END_VAR
M_Read := THIS^.stSeqCtrlGeneral.eActiveSeqState = E_SEQ_GENERAL.DONE;

// Assign input
THIS^.udiDBID := udiDBID;
THIS^.sTableName := sTableName;
THIS^.sDBSymbolName := sDBSymbolName;
THIS^.eOrderBy := eOrderBy;
THIS^.eOrderType := eOrderType;
THIS^.nStartIndex := nStartIndex;
THIS^.nRecordCount := nRecordCount;
THIS^.pData2 := pData2;
THIS^.cbData := cbData;

// General
IF THIS^.stSeqCtrlGeneral.eActiveSeqState = E_SEQ_GENERAL.READY THEN
  THIS^.eNextSeq := E_SEQ_DATABASE.READ;
  THIS^.stSeqCtrlGeneral.eActiveSeqState := E_SEQ_GENERAL.EXECUTE;
END_IF

// Example
(*
VAR
    fbPLCDBRead    : FB_PLCDBReadEvt (sNetID := '', tTimeout := T#5S);
    ReadStruct     : ST_StandardRecord;
    tcMessage      : I_TcMessage;
END_VAR

------------------------------------------------------------------------

IF fbPLCDBRead.Read(
    hDBID:= 1, 
    sTableName:= 'MyTable_WithLReal', 
    sDBSymbolName:= 'MyValue', 
    eOrderBy:= E_OrderColumn.ID, 
    eOrderType:= E_OrderType.DESC, 
    nStartIndex:= 0, 
    nRecordCount:= 1, 
    pData:= ADR(ReadStruct), 
    cbData:= SIZEOF(ReadStruct))
THEN
    IF fbPLCDBRead.bError THEN
        tcMessage := fbPLCDBRead.ipTcResult;
        nState := 255; 
    ELSE
        nState := 0;
    END_IF
END_IF
*)
END_METHOD

METHOD M_ReadStruct : BOOL

VAR_INPUT
  /// Indicates the ID of the database to be used.
  udiDBID:                    UDINT;
  /// Name of the table that is to be read.
  sTableName:                 T_MaxString;
  /// Address of the array containing the column name to be read.
  pColumnNames:               POINTER TO ARRAY [0..MAX_DBCOLUMNS] OF STRING(50);
  /// Length of the column name array
  cbColumnNames:              UDINT;
  /// Name the sorting column
  sOrderByColumn:             STRING(50);
  /// Sorting direction (ASC or DESC)
  eOrderType:                 E_OrderType;
  /// Indicates the index of the first record to be read.
  nStartIndex:                UDINT;
  /// Indicates the number of records to be read.
  nRecordCount:               UDINT;
  /// Address of the structure array into which the records are to be written.
  pData:                      POINTER TO BYTE;
  /// Indicates the size of the structure array in bytes.
  cbData:                     UDINT;
END_VAR
VAR
  
END_VAR
M_ReadStruct := THIS^.stSeqCtrlGeneral.eActiveSeqState = E_SEQ_GENERAL.DONE;

// Assign input
THIS^.udiDBID := udiDBID;
THIS^.sTableName := sTableName;
THIS^.pColumnNames := pColumnNames;
THIS^.cbColumnNames := cbColumnNames;
THIS^.sOrderByColumn := sOrderByColumn;
THIS^.eOrderType := eOrderType;
THIS^.nStartIndex := nStartIndex;
THIS^.nRecordCount := nRecordCount;
THIS^.pData := pData;
THIS^.cbData := cbData;

// General
IF THIS^.stSeqCtrlGeneral.eActiveSeqState = E_SEQ_GENERAL.READY THEN
  THIS^.eNextSeq := E_SEQ_DATABASE.READ_STRUCT;
  THIS^.stSeqCtrlGeneral.eActiveSeqState := E_SEQ_GENERAL.EXECUTE;
END_IF

// Example
(*
VAR
    fbPLCDBRead    : FB_PLCDBReadEvt (sNetID := '', tTimeout := T#5S);
    myCustomStruct : ST_Record;
    tcMessage      : I_TcMessage;
END_VAR

------------------------------------------------------------------------

TYPE ST_Record :
STRUCT
    nID        : LINT;
    dtTimestamp: DATE_AND_TIME;
    sName      : STRING;
    nSensor1   : LREAL;
    nSensor2   : LREAL;
END_STRUCT
END_TYPE

--------------------------------------------------------------------------

// set columnnames
ColumnNames[0] := 'ID';
ColumnNames[1] := 'Timestamp';
ColumnNames[2] := 'Name';
ColumnNames[3] := 'Sensor1';
ColumnNames[4] := 'Sensor2';

IF fbPLCDBRead.ReadStruct(
    hDBID:= 1, 
    sTableName:= 'MyTable_Struct', 
    pColumnNames:= ADR(ColumnNames), 
    cbColumnNames:= SIZEOF(ColumnNames), 
    sOrderByColumn:= ColumnNames[0], 
    eOrderType:= E_OrderType.DESC, 
    nStartIndex:= 0, 
    nRecordCount:= 1, 
    pData:= ADR(myCustomStruct), 
    cbData:= SIZEOF(myCustomStruct))
THEN
    IF fbPLCDBRead.bError THEN
        tcMessage:= fbPLCDBRead.ipTcResult;
        nState := 255; 
    ELSE
        nState := 0;
    END_IF
END_IF
*)
END_METHOD

METHOD M_Reset : BOOL
M_Reset := THIS^.stSeqCtrlGeneral.eActiveSeqState = E_SEQ_GENERAL.DONE;

// General
IF THIS^.stSeqCtrlGeneral.eActiveSeqState = E_SEQ_GENERAL.READY THEN
  THIS^.eNextSeq := E_SEQ_DATABASE.INIT;
  THIS^.stSeqCtrlGeneral.eActiveSeqState := E_SEQ_GENERAL.EXECUTE;
END_IF
END_METHOD

(*=== Method: M_Run  ============================================

 @brief: Here is the global code (Timer, Event, Flange,...)*)
METHOD M_Run
END_METHOD

METHOD M_SetReady : BOOL
VAR_INPUT
END_VAR
M_SetReady := TRUE
              AND THIS^.stSeqCtrlGeneral.eActiveSeqState = E_SEQ_GENERAL.READY
              AND THIS^.eSeq = E_SEQ_DATABASE.BASE;

THIS^.stSeqCtrlGeneral.eActiveSeqState := E_SEQ_GENERAL.READY;
THIS^.eNextSeq := E_SEQ_DATABASE.BASE;
END_METHOD

METHOD M_TableExistCheck : BOOL
VAR_INPUT
  /// Indicates the ID of the database to be used.
  udiDBID:                    UDINT;
  /// Name of the table that is to be read.
  sTableName:                 T_MaxString;
END_VAR
VAR_OUTPUT
  /// Result
  bResult:                    BOOL;
END_VAR
M_TableExistCheck := THIS^.stSeqCtrlGeneral.eActiveSeqState = E_SEQ_GENERAL.DONE;

// Assign input
THIS^.udiDBID := udiDBID;
THIS^.sTableName := sTableName;
THIS^.sCmd := CONCAT('SELECT * FROM $'', sTableName);
THIS^.sCmd := CONCAT(THIS^.sCmd, '$'');
THIS^.pSQLCmd := ADR(THIS^.sCmd);
THIS^.cbSQLCmd := SIZEOF(THIS^.sCmd);

// Assign output
bResult := THIS^.bResult;

// General
IF THIS^.stSeqCtrlGeneral.eActiveSeqState = E_SEQ_GENERAL.READY THEN
  THIS^.eNextSeq := E_SEQ_DATABASE.TABLE_EXIST_CHECK;
  THIS^.stSeqCtrlGeneral.eActiveSeqState := E_SEQ_GENERAL.EXECUTE;
END_IF
END_METHOD

METHOD M_Write : BOOL

VAR_INPUT
  /// Indicates the ID of the database to be used.
  udiDBID:            UDINT;
  /// Name of the table that is to be write.
  sTableName:         T_MaxString;
  /// Address of the variable to be logged in the standard table structure.
  pValue:             POINTER TO BYTE;
  /// Length of the variable to be logged.
  cbValue:            UDINT;
  /// Name that is logged in the table.
  sDBSymbolName:      STRING;
  /// Indicates the write mode. (append, update, ring buffer)
  eDBWriteMode:       E_WriteMode;
  /// Additional parameter(s) for the "ring buffer" write mode.
  nRingBuffParameter: UDINT;
END_VAR
M_Write := THIS^.stSeqCtrlGeneral.eActiveSeqState = E_SEQ_GENERAL.DONE;

// Assign input
THIS^.udiDBID := udiDBID;
THIS^.sTableName := sTableName;
THIS^.pValue := pValue;
THIS^.cbValue := cbValue;
THIS^.sDBSymbolName := sDBSymbolName;
THIS^.eDBWriteMode := eDBWriteMode;
THIS^.nRingBuffParameter := nRingBuffParameter;

// General
IF THIS^.stSeqCtrlGeneral.eActiveSeqState = E_SEQ_GENERAL.READY THEN
  THIS^.eNextSeq := E_SEQ_DATABASE.WRITE;
  THIS^.stSeqCtrlGeneral.eActiveSeqState := E_SEQ_GENERAL.EXECUTE;
END_IF

// Example
(*
VAR
    fbPLCDBWrite    : FB_PLCDBWriteEvt(sNetID := '', tTimeout := T#5S);
    myValue         : LREAL := 43.23;
    tcMessage       : I_TcMessage;
END_VAR

------------------------------------------------------------------------

IF fbPLCDBWrite.Write(
    hDBID:= 1, 
    sTableName:= 'myTable_WithLReal',
    pValue:= ADR(myValue), 
    cbValue:= SIZEOF(myValue), 
    sDBSymbolName:= 'MyValue', 
    eDBWriteMode:= E_WriteMode.eADS_TO_DB_RingBuff_Count, 
    nRingBuffParameter:= 3) 
THEN
    IF fbPLCDBWrite.bError THEN
        tcMessage := fbPLCDBWrite.ipTcResult;
        nState := 255; 
    ELSE
        nState := 0; 
    END_IF
END_IF
*)
END_METHOD

METHOD M_WriteBySymbol : BOOL

VAR_INPUT
  /// Indicates the ID of the database to be used.
  udiDBID:            UDINT;
  /// Name of the table that is to be write.
  sTableName:         T_MaxString;
  /// ADS device from which a symbol is to be logged in the standard table structure.
  stADSDevice:        ST_ADSDevice;
  /// Symbol name of the variable to be written
  stSymbol:           ST_Symbol;
  /// Indicates the write mode. (append, update, ring buffer)
  eDBWriteMode:       E_WriteMode;
  /// Additional parameter(s) for the "ring buffer" write mode.
  nRingBuffParameter: UDINT;
END_VAR
M_WriteBySymbol := THIS^.stSeqCtrlGeneral.eActiveSeqState = E_SEQ_GENERAL.DONE;

// Assign input
THIS^.udiDBID := udiDBID;
THIS^.sTableName := sTableName;
THIS^.stADSDevice := stADSDevice;
THIS^.stSymbol := stSymbol;
THIS^.eDBWriteMode := eDBWriteMode;
THIS^.nRingBuffParameter := nRingBuffParameter;



// General
IF THIS^.stSeqCtrlGeneral.eActiveSeqState = E_SEQ_GENERAL.READY THEN
  THIS^.eNextSeq := E_SEQ_DATABASE.WRITE_BY_SYMBOL;
  THIS^.stSeqCtrlGeneral.eActiveSeqState := E_SEQ_GENERAL.EXECUTE;
END_IF

// Example
(*
VAR
    fbPLCDBWrite    :  FB_PLCDBWriteEvt(sNetID := '', tTimeout := T#5S);
    myValue         :  LREAL := 43.23;
    myAdsDevice     :  ST_ADSDevice;
    mySymbol        :  ST_Symbol;
    tcMessage       :  I_TcMessage;
END_VAR

------------------------------------------------------------------------

// Set ADSDevice Information
myAdsDevice.sDevNetID     := '127.0.0.1.1.1';
myAdsDevice.nDevPort      := 851;
myAdsDevice.eADSRdWrtMode := E_ADSRdWrtMode.bySymbolName; 
myAdsDevice.tTimeout      := T#5S; 

// Set Symbol Information
mySymbol.eDataType        := E_PLCDataType.eType_LREAL;
mySymbol.sDBSymbolName    := 'MySymbol';
mySymbol.sSymbolName      := 'MAIN.myValue';
mySymbol.nBitSize         := 8;

// Call Functionblock
IF fbPLCDBWrite.WriteBySymbol(
    hDBID:= 1, 
    sTableName:= 'myTable_WithLReal', 
    stADSDevice:= myAdsDevice, 
    stSymbol:= mySymbol, 
    eDBWriteMode:= E_WriteMode.eADS_TO_DB_Append, 
    nRingBuffParameter:= 1) 
THEN
    IF fbPLCDBWrite.bError THEN
        tcMessage := fbPLCDBWrite.ipTcResult;
        nState := 255; 
    ELSE
        nState := 0;
    END_IF
END_IF
*)
END_METHOD

METHOD M_WriteStruct : BOOL
VAR_INPUT
  /// Indicates the ID of the database to be used.
  udiDBID:        UDINT;
  /// Name of the table that is to be write.
  sTableName:     T_MaxString;
  /// Address of a structure that is to be logged in a freely selectable table structure.
  pRecord:        POINTER TO BYTE;
  /// Length of the structure to be written
  cbRecord:       UDINT;
  /// Address of the array containing the column name to be filled.
  pColumnNames:   POINTER TO ARRAY [0..MAX_DBCOLUMNS] OF STRING(50);
  /// Length of the column name array
  cbColumnNames:  UDINT;
END_VAR
M_WriteStruct := THIS^.stSeqCtrlGeneral.eActiveSeqState = E_SEQ_GENERAL.DONE;

// Assign input
THIS^.udiDBID := udiDBID;
THIS^.sTableName := sTableName;
THIS^.pRecord := pRecord;
THIS^.cbRecord := cbRecord;
THIS^.pColumnNames := pColumnNames;
THIS^.cbColumnNames := cbColumnNames;

// General
IF THIS^.stSeqCtrlGeneral.eActiveSeqState = E_SEQ_GENERAL.READY THEN
  THIS^.eNextSeq := E_SEQ_DATABASE.WRITE_STRUCT;
  THIS^.stSeqCtrlGeneral.eActiveSeqState := E_SEQ_GENERAL.EXECUTE;
END_IF

// Example
(*
VAR
    fbPLCDBWrite    :  FB_PLCDBWriteEvt(sNetID := '', tTimeout := T#5S);
    myRecord        :  ST_Record;
    ColumnNames     :  ARRAY[0..4] OF STRING(50);
    
    systime         :  GETSYSTEMTIME;
    currentTime     :  T_FILETIME;
    tcMessage       :  I_TcMessage;
END_VAR

------------------------------------------------------------------------

TYPE ST_Record :
STRUCT
    nID        : LINT;
    dtTimestamp: DATE_AND_TIME;
    sName      : STRING;
    nSensor1   : LREAL;
    nSensor2   : LREAL;
END_STRUCT
END_TYPE

------------------------------------------------------------------------

// set Values
systime(timeLoDw => currentTime.dwLowDateTime, timeHiDW => currentTime.dwHighDateTime );
myRecord.dtTimestamp := FILETIME_TO_DT(currentTime);
myRecord.sName       := 'MyStructVal';
myRecord.nSensor1    := 12.34;
myRecord.nSensor2    := 102.5;

// set columnnames
ColumnNames[0] := 'ID';
ColumnNames[1] := 'Timestamp';
ColumnNames[2] := 'Name';
ColumnNames[3] := 'Sensor1';
ColumnNames[4] := 'Sensor2';

// Call Functionblock
IF fbPLCDBWrite.WriteStruct(
    hDBID:= 1, 
    sTableName:= 'myTable_Struct', 
    pRecord:= ADR(myRecord), 
    cbRecord:= SIZEOF(myRecord), 
    pColumnNames:= ADR(ColumnNames) , 
    cbColumnNames:= SIZEOF(ColumnNames))
THEN
    IF fbPLCDBWrite.bError THEN
        tcMessage := fbPLCDBWrite.ipTcResult;
        nState := 255; 
    ELSE
        nState := 0;
    END_IF
END_IF
*)
END_METHOD

PROPERTY P_Connected : BOOL
GET
P_Connected := THIS^.fbSQLDatabase.bConnected;
END_GET
END_PROPERTY

{warning 'Eigenschaftenimplementierung hinzufügen'}
PROPERTY P_Error : BOOL
GET
P_Error := THIS^.stSeqCtrlGeneral.eActiveSeqState = E_SEQ_GENERAL.ERROR;
END_GET
END_PROPERTY

{warning 'Eigenschaftenimplementierung hinzufügen'}
(*=== Property: P_Event  ============================================

 @param [set]: 	Set the Structure "ST_EVENT" from another Object
 @param [get]: 	Return the Structure "ST_EVENT", it contains the actual 
					event of the Object *)
PROPERTY P_Event : GenLib.ST_EVENT
GET
END_GET
SET
END_SET
END_PROPERTY

{warning 'Eigenschaftenimplementierung hinzufügen'}
(*=== Property: P_FullObjectPath  ============================================

 @param [set]: 	Set the Object Path (Clear String of Object)
 @param [get]: 	Return the Objectpath *)
PROPERTY P_FullObjectPath : STRING
GET
P_FullObjectPath:= THIS^.strFullObjectPath;
END_GET
SET
THIS^.strFullObjectPath:=P_FullObjectPath;
END_SET
END_PROPERTY

{warning 'Eigenschaftenimplementierung hinzufügen'}
(*=== Property: P_Global_Ack  ============================================

 @param [set]: 	Set the Bit for Ack from another Object
 @param [get]: 	Return the state of Ack Bit*)
PROPERTY P_Global_Ack : BOOL
GET
END_GET
SET
END_SET
END_PROPERTY

{warning 'Eigenschaftenimplementierung hinzufügen'}
(*=== Property: P_GlobalID  ============================================

 @param [set]: 	-
 @param [get]: 	Return the string of instance path*)
PROPERTY P_GlobalID : STRING
GET
P_GlobalID:= THIS^.strInstancePath;
END_GET
END_PROPERTY

END_FUNCTION_BLOCK

// ---- MODULE/FREQUENCE/POU/FB_FREQENCE.TcPOU
{attribute 'reflection'} 
{attribute 'no_explicit_call' := 'do not call this POU directly'} 
FUNCTION_BLOCK PUBLIC FB_FREQENCE IMPLEMENTS  I_FREQ_GEN
VAR_INPUT
END_VAR
VAR_OUTPUT
END_VAR
VAR
	{attribute 'instance-path'} 
    {attribute 'noinit'} 
	strInstancePath: STRING;
	strFullObjectPath: STRING;
	stEvent: ST_EVENT;
	bAck: BOOL;
	
	iStep:		INT:=0;
	tonLow:		TON;
	tonHigh:	TON;
	tFreq:		TIME;
	bState:		BOOL;
	iFreqence:	INT;
	fTrig:		F_TRIG;
	rTrig:		R_TRIG;
END_VAR

(*=== Method: M_Run  ============================================

 @brief: Here is the global code (Timer, Event, Flange,...)*)
METHOD M_Run
tFreq := TO_TIME(TO_REAL(1000 * iFreqence) / 2);

CASE iStep OF
0:;	IF tonLow.Q THEN iStep := 1; END_IF;
1:;	IF tonHigh.Q THEN iStep := 0; END_IF;
ELSE
	iStep := 0;
END_CASE

tonHigh(IN:=(iStep=1), PT:= tFreq);
tonLow(IN:= (iStep=0), PT:= tFreq);

bState:=(iStep>=1);

fTrig(CLK:=bState);
rTrig(CLK:=bState);
END_METHOD

METHOD M_SetFrequence : bool
VAR_INPUT
	iFreqence: INT;
END_VAR
M_SetFrequence := TRUE;

THIS^.iFreqence := iFreqence;
END_METHOD

(*=== Property: P_Event  ============================================

 @param [set]: 	Set the Structure "ST_EVENT" from another Object
 @param [get]: 	Return the Structure "ST_EVENT", it contains the actual 
					event of the Object *)
PROPERTY P_Event : GenLib.ST_EVENT
GET
P_Event:=stEvent;
END_GET
SET
stEvent:=P_Event;
END_SET
END_PROPERTY

PROPERTY P_FTrig : BOOL
GET
P_FTrig:=THIS^.fTrig.Q;
END_GET
END_PROPERTY

(*=== Property: P_FullObjectPath  ============================================

 @param [set]: 	Set the Object Path (Clear String of Object)
 @param [get]: 	Return the Objectpath *)
PROPERTY P_FullObjectPath : STRING
GET
P_FullObjectPath:= THIS^.strFullObjectPath;
END_GET
SET
THIS^.strFullObjectPath:=P_FullObjectPath;
END_SET
END_PROPERTY

(*=== Property: P_Global_Ack  ============================================

 @param [set]: 	Set the Bit for Ack from another Object
 @param [get]: 	Return the state of Ack Bit*)
PROPERTY P_Global_Ack : BOOL
GET
P_Global_Ack:=THIS^.bAck;
END_GET
SET
THIS^.bAck:=P_Global_Ack;
END_SET
END_PROPERTY

(*=== Property: P_GlobalID  ============================================

 @param [set]: 	-
 @param [get]: 	Return the string of instance path*)
PROPERTY P_GlobalID : STRING
GET
P_GlobalID:= THIS^.strInstancePath;
END_GET
END_PROPERTY

PROPERTY P_RTrig : BOOL
GET
P_RTrig := THIS^.rTrig.Q;
END_GET
END_PROPERTY

PROPERTY P_State : BOOL
GET
P_State:=THIS^.bState;
END_GET
END_PROPERTY

END_FUNCTION_BLOCK

// ---- MODULE/GENERAL/F_Lineare_Regression.TcPOU
FUNCTION F_Lineare_Regression : stRampAnalytic
VAR_IN_OUT
	Messwerte:          ARRAY[*] OF stMesswerte;
	uiStart: 	          UINT;	
	uiEnd: 		          UINT; 	///Bei 0 gilt Upper Bound
END_VAR
VAR
	i: 					        DINT;
	diLow: 				      DINT;
	diHigh: 			      DINT;
	rMittelwert: 		    stMesswerte;
	lrSteigung: 		    LREAL;
	lrAchsenabschnitt: 	LREAL;
	lrTempY_s: 			    LREAL;
	lrZaehlerMw: 		    LREAL;
	lrNennerMw: 		    LREAL;
	lrSumSqrtY_Ys:		  LREAL;
	lrSumSqrtY_Yd:		  LREAL;
	lrSqrtR:			      LREAL;
	
	stOut:				      stRampAnalytic;
	bFault:             BOOL;
END_VAR

F_Lineare_Regression.lrGain := 0;
F_Lineare_Regression.lrOffset := 0;
F_Lineare_Regression.lrExp2R := -1;
diLow := LOWER_BOUND(Messwerte, 1);
diHigh := UPPER_BOUND(Messwerte, 1);
IF uiEnd > 0 THEN
	diLow := uiStart;
	diHigh := uiEnd;
END_IF 
rMittelwert.X := 0;
rMittelwert.Y := 0;
//Mittelwert ermitteln
FOR i := diLow TO diHigh DO
	rMittelwert.X := rMittelwert.X + Messwerte[i].X;
	rMittelwert.Y := rMittelwert.Y + Messwerte[i].Y;
END_FOR
	IF (DINT_TO_REAL(diHigh - diLow) + 1) <> 0 THEN
	rMittelwert.X := rMittelwert.X / (DINT_TO_REAL(diHigh - diLow) + 1);
	rMittelwert.Y := rMittelwert.Y / (DINT_TO_REAL(diHigh - diLow) + 1);
ELSE
	bFault := TRUE;	
END_IF

//Steigung = Mittelwert X durch Mittelwert Y


lrZaehlerMw := 0;
lrNennerMw := 0;

FOR i:=diLow TO diHigh DO
	lrZaehlerMw :=	lrZaehlerMw + (Messwerte[i].X - rMittelwert.X) * (Messwerte[i].Y - rMittelwert.Y);
	//lrNennerMw:=	lrNennerMw+		(basic.expn((Messwerte[i].X-rMittelwert.X),2));
END_FOR
//lrZaehlerMw:=	lrZaehlerMw	/(DINT_TO_REAL(diHigh-diLow)+0);
//lrNennerMw:=	lrNennerMw	/(DINT_TO_REAL(diHigh-diLow)+0);


//Steigung = 
IF lrNennerMw <> 0 THEN
	lrSteigung := lrZaehlerMw / lrNennerMw;
ELSE
	bFault := TRUE;
END_IF
lrAchsenabschnitt := rMittelwert.Y - (lrSteigung * rMittelwert.X);
(*
FOR i:=diLow TO diHigh DO
	lrTempY_s:=					(Messwerte[i].X*lrSteigung)+lrAchsenabschnitt;
	Messwerte[i].sqr_Y_Ys:=		basic.EXPN((Messwerte[i].Y-lrTempY_s),2);
	
	Messwerte[i].SQR_Y_Yd:=		basic.EXPN((Messwerte[i].Y-rMittelwert.Y),2);
END_FOR
*)
lrSumSqrtY_Ys := 0;
lrSumSqrtY_Yd := 0;
(*
FOR i:=diLow TO diHigh DO
	lrSumSqrtY_Ys:=lrSumSqrtY_Ys+Messwerte[i].sqr_Y_Ys;
	lrSumSqrtY_Yd:=lrSumSqrtY_Yd+Messwerte[i].SQR_Y_Yd;
END_FOR
*)
FOR i := diLow TO diHigh DO
	lrTempY_s := (Messwerte[i].X * lrSteigung) + lrAchsenabschnitt;
	//lrSumSqrtY_Ys:=	lrSumSqrtY_Ys+	basic.EXPN((Messwerte[i].Y-lrTempY_s),2);
	
	//lrSumSqrtY_Yd:=	lrSumSqrtY_Yd+	basic.EXPN((Messwerte[i].Y-rMittelwert.Y),2);
END_FOR

IF lrSumSqrtY_Yd <> 0 THEN
	lrSqrtR := 1 - (lrSumSqrtY_Ys / lrSumSqrtY_Yd);
ELSE
	bFault := TRUE;
END_IF
IF NOT bFault THEN
	F_Lineare_Regression.lrGain := lrSteigung;
	F_Lineare_Regression.lrOffset := lrAchsenabschnitt;
	F_Lineare_Regression.lrExp2R := lrSqrtR;
END_IF

END_FUNCTION

// ---- MODULE/GENERAL/F_RangeSetpoint.TcPOU
FUNCTION F_RangeSetpoint : BOOL
VAR_INPUT
	lrSetpoint: LREAL;
	lrActValue: LREAL;
	lrRangePercent: LREAL;
END_VAR
VAR
	lrTempSetpointUp: LREAL;
	lrTempSetpointDown: LREAL;
END_VAR

F_RangeSetpoint:=FALSE;

lrTempSetpointDown:=lrSetpoint-(lrSetpoint*(lrRangePercent/100.0));
lrTempSetpointUp:=lrSetpoint+(lrSetpoint*(lrRangePercent/100.0));

IF (lrActValue>=lrTempSetpointDown) AND (lrActValue<=lrTempSetpointUp) THEN
	F_RangeSetpoint:=TRUE;
END_IF

END_FUNCTION

// ---- MODULE/GENERAL/INPUTS/POU/FB_BINARY_SWITCH_SENS.TcPOU
FUNCTION_BLOCK FB_BINARY_SWITCH_SENS IMPLEMENTS  I_BINARY_SWITCH_SENS
VAR_INPUT
END_VAR
VAR_OUTPUT
END_VAR
VAR
		
	itfOpMode:										I_OP_MODE;
	{attribute 'instance-path'} 
    {attribute 'noinit'} 
	strInstancePath:								STRING;
	strFullObjectPath:								STRING;
	stEvent:										ST_EVENT;
	bAck:											BOOL;
	
	bSwitch 										AT %I*: BOOL;
	bNC:											BOOL;
	fbEventLogger:									FB_TcEventLogger;
	                                				
	strSymName:										STRING;
	iStepCase:										INT;
	strMessage:										STRING;
	bSensingON:										BOOL;
END_VAR

strFullObjectPath:=F_CreateIdString(THIS^);


stEvent.bEventActive:=FALSE;
IF THIS^.bSensingON AND P_Active THEN
	fbEventLogger.GetAlarm(eventClass:= TC_EVENT_CLASSES.TcSystemEventClass,
							nEventID:=1,
							ipSourceInfo:=TRUE,
							fbAlarm:=TRUE);
END_IF



//Überwachung Eingang
CASE iStepCase OF
	
	0://SENSING Deaktiviert
	
	
	1://SENSING Aktiviert
		
		
	
	
	re
END_CASE

METHOD FB_init : BOOL
VAR_INPUT
	bInitRetains : BOOL; // if TRUE, the retain variables are initialized (warm start / cold start)
	bInCopyCode : BOOL;  // if TRUE, the instance afterwards gets moved into the copy code (online change)
	itfOpMode:			I_OP_MODE;
	bInNC: 				BOOL;///NC:=true; NO:= false
	strMessage:			STRING;
	bSensingON:			BOOL;
END_VAR
THIS^.itfOpMode:=	itfOpMode;
THIS^.bNC:=			bInNC;
THIS^.strMessage:=	strMessage;
THIS^.bSensingON:=	bSensingON;
END_METHOD

(*=== Method: M_Run  ============================================

 @brief: Here is the global code (Timer, Event, Flange,...)*)
METHOD M_Run
END_METHOD

METHOD M_START_SENS : BOOL
VAR_INPUT
	bState	: BOOL;
	tDelay	: TIME;
	eEventType	: GenLib.ENUM_EVENT_TYPE;
END_VAR
IF THIS^.iStepCase=0 THEN
	THIS^.iStepCase:=1;
END_IF
END_METHOD

METHOD M_STOP_SENS : BOOL
END_METHOD

PROPERTY P_Active : BOOL
GET
IF bNC THEN
	P_ACTIVE:= NOT bSwitch;
ELSE
	P_ACTIVE:= bSwitch;
END_IF
END_GET
END_PROPERTY

(*=== Property: P_Event  ============================================

 @param [set]: 	Set the Structure "ST_EVENT" from another Object
 @param [get]: 	Return the Structure "ST_EVENT", it contains the actual 
					event of the Object *)
PROPERTY P_Event : GenLib.ST_EVENT
GET
P_Event:=stEvent;
END_GET
SET
stEvent:=P_Event;
END_SET
END_PROPERTY

(*=== Property: P_FullObjectPath  ============================================

 @param [set]: 	Set the Object Path (Clear String of Object)
 @param [get]: 	Return the Objectpath *)
PROPERTY P_FullObjectPath : STRING
GET
P_FullObjectPath:= THIS^.strFullObjectPath;
END_GET
SET
END_SET
END_PROPERTY

(*=== Property: P_Global_Ack  ============================================

 @param [set]: 	Set the Bit for Ack from another Object
 @param [get]: 	Return the state of Ack Bit*)
PROPERTY P_Global_Ack : BOOL
GET
P_Global_Ack:=THIS^.bAck;
END_GET
SET
THIS^.bAck:=P_Global_Ack;
END_SET
END_PROPERTY

{warning 'Eigenschaftenimplementierung hinzufügen'}
(*=== Property: P_GlobalID  ============================================

 @param [set]: 	-
 @param [get]: 	Return the string of instance path*)
PROPERTY P_GlobalID : STRING
GET
P_GlobalID:= THIS^.strInstancePath;
END_GET
END_PROPERTY

PROPERTY P_No_Nc : BOOL
GET
P_No_Nc:= not THIS^.bNC;
END_GET
END_PROPERTY

PROPERTY P_On : BOOL
GET
P_ON:= bSwitch;
END_GET
END_PROPERTY

PROPERTY P_STATE_SENS : BOOL
GET
END_GET
END_PROPERTY

END_FUNCTION_BLOCK

// ---- MODULE/GENERAL/SIMU_ANALOG_IN/FB_SIMU_ANALOG_IN.TcPOU
{attribute 'reflection'} 
FUNCTION_BLOCK FB_SIMU_ANALOG_IN IMPLEMENTS  I_SIMU_ANALOG_IN
VAR_INPUT
END_VAR
VAR_OUTPUT
END_VAR
VAR
	lrSetPoint: LREAL;
	{attribute 'instance-path'} 
    {attribute 'noinit'} 
	strInstancePath: STRING;
	strFullObjectPath: STRING;
END_VAR

{warning 'Methodenimplementierung hinzufügen'}
(*=== Method: M_Run  ============================================

 @brief: Here is the global code (Timer, Event, Flange,...)*)
METHOD M_Run
THIS^.strFullObjectPath:= F_CreateIdString(THIS^);
END_METHOD

{warning 'Eigenschaftenimplementierung hinzufügen'}
(*=== Property: P_Event  ============================================

 @param [set]: 	Set the Structure "ST_EVENT" from another Object
 @param [get]: 	Return the Structure "ST_EVENT", it contains the actual 
					event of the Object *)
PROPERTY P_Event : GenLib.ST_EVENT
GET
END_GET
SET
END_SET
END_PROPERTY

{warning 'Eigenschaftenimplementierung hinzufügen'}
(*=== Property: P_FullObjectPath  ============================================

 @param [set]: 	Set the Object Path (Clear String of Object)
 @param [get]: 	Return the Objectpath *)
PROPERTY P_FullObjectPath : STRING
GET
P_FullObjectPath:= THIS^.strFullObjectPath;
END_GET
SET
THIS^.strFullObjectPath:=P_FullObjectPath;
END_SET
END_PROPERTY

{warning 'Eigenschaftenimplementierung hinzufügen'}
(*=== Property: P_Global_Ack  ============================================

 @param [set]: 	Set the Bit for Ack from another Object
 @param [get]: 	Return the state of Ack Bit*)
PROPERTY P_Global_Ack : BOOL
GET
END_GET
SET
END_SET
END_PROPERTY

{warning 'Eigenschaftenimplementierung hinzufügen'}
(*=== Property: P_GlobalID  ============================================

 @param [set]: 	-
 @param [get]: 	Return the string of instance path*)
PROPERTY P_GlobalID : STRING
GET
P_GlobalID:= THIS^.strInstancePath;
END_GET
END_PROPERTY

{warning 'Eigenschaftenimplementierung hinzufügen'}
PROPERTY P_SETPOINT : LREAL
SET
lrSetPoint:=P_SETPOINT;
END_SET
END_PROPERTY


PROPERTY P_VALUE : LREAL
GET
P_VALUE:=lrSetPoint;
END_GET
END_PROPERTY

END_FUNCTION_BLOCK

// ---- MODULE/HMI/POU/FB_HMI_CTRL.TcPOU
FUNCTION_BLOCK FB_HMI_CTRL IMPLEMENTS I_HMI_CTRL
VAR_INPUT
END_VAR
VAR_OUTPUT
END_VAR
VAR
  strInstancePath:                STRING;
	strFullObjectPath:              STRING;
  strErrorMsg:                    STRING := '';
  bInHP:                          BOOL;
	stEvent:                        ST_EVENT;
	bAck:                           BOOL;
	itfOpMode:			                I_OP_MODE;
  
  //HMI Start
	fbHmiStart:							  NT_StartProcess;
	bHmiStart:							  BOOL;
	//HMI Kill
	fbTaskKill:							  NT_StartProcess;
	bTaskKill:							  BOOL;
	//Shutdown Windows
	fbShutdown:							  NT_StartProcess;
	bShutdown:							  BOOL;
	//Reboot Windows
	fbReboot:							    NT_StartProcess;
	bReboot:							    BOOL;
	//Windows Keyboard
	fbWinKeyboard:						NT_StartProcess;
	bWinKeyboard:						  BOOL;
END_VAR

fbHmiStart(
	NETID:= '', 
	PATHSTR:= 'C:\Program Files (x86)\Microsoft\Edge\Application\msedge.exe', 
	DIRNAME:= 'C:\Program Files (x86)\Microsoft\Edge\Application', 
	COMNDLINE:= '--kiosk http://Administrator:1@127.0.0.1:1010 --edge-kiosk-type=fullscreen', 
	START:= bHmiStart, 
	TMOUT:= T#25S, 
	BUSY=> , 
	ERR=> , 
	ERRID=> );
IF fbHmiStart.BUSY THEN
	bHmiStart:=FALSE;
END_IF

fbTaskKill(
	NETID:= '', 
	PATHSTR:= 'C:\Scripts\CloseHMI.bat', 
	DIRNAME:= 'C:\Scripts', 
	COMNDLINE:= '', 
	START:= bTaskKill, 
	TMOUT:= T#5S, 
	BUSY=> , 
	ERR=> , 
	ERRID=> );
IF fbTaskKill.BUSY THEN
	bTaskKill:=FALSE;
END_IF

fbWinKeyboard(
	NETID:= '', 
	PATHSTR:= 'C:\Scripts\Keyboard.bat', 
	DIRNAME:= 'C:\Scripts', 
	COMNDLINE:= '', 
	START:= bWinKeyboard, 
	TMOUT:= T#5S, 
	BUSY=> , 
	ERR=> , 
	ERRID=> );
IF fbWinKeyboard.BUSY THEN
	bWinKeyboard:=FALSE;
END_IF

fbShutdown(
	NETID:= '', 
	PATHSTR:= 'C:\Scripts\Shutdown.bat', 
	DIRNAME:= 'C:\Scripts', 
	COMNDLINE:= '', 
	START:= bShutdown, 
	TMOUT:= T#30S, 
	BUSY=> , 
	ERR=> , 
	ERRID=> );
IF fbShutdown.BUSY THEN
	bShutdown:=FALSE;
END_IF

fbReboot(
	NETID:= '', 
	PATHSTR:= 'C:\Scripts\Reboot.bat', 
	DIRNAME:= 'C:\Scripts', 
	COMNDLINE:= '', 
	START:= bReboot, 
	TMOUT:= T#30S, 
	BUSY=> , 
	ERR=> , 
	ERRID=> );
IF fbReboot.BUSY THEN
	bReboot:=FALSE;
END_IF

METHOD FB_init : BOOL
VAR_INPUT
	bInitRetains : BOOL; // if TRUE, the retain variables are initialized (warm start / cold start)
	bInCopyCode : BOOL;  // if TRUE, the instance afterwards gets moved into the copy code (online change)
END_VAR
END_METHOD

METHOD M_CloseHMI : BOOL
bTaskKill := TRUE;
END_METHOD

METHOD M_HideWinKeyboard : BOOL
END_METHOD

METHOD M_PCReboot : BOOL
bReboot := TRUE;
END_METHOD

METHOD M_PCShutdown : BOOL
bShutdown := TRUE;
END_METHOD

{warning 'Methodenimplementierung hinzufügen'}
(*=== Method: M_Run  ============================================

 @brief: Here is the global code (Timer, Event, Flange,...)*)
METHOD M_Run
END_METHOD

{warning 'Methodenimplementierung hinzufügen'}
METHOD M_SetReady : BOOL
END_METHOD

METHOD M_ShowWinKeyboard : BOOL
bWinKeyboard := TRUE;
END_METHOD

METHOD M_StartHMI : BOOL
bHmiStart := TRUE;
END_METHOD

{warning 'Eigenschaftenimplementierung hinzufügen'}
PROPERTY P_ErrorMsg : STRING
GET
END_GET
SET
END_SET
END_PROPERTY

{warning 'Eigenschaftenimplementierung hinzufügen'}
(*=== Property: P_Event  ============================================

 @param [set]: 	Set the Structure "ST_EVENT" from another Object
 @param [get]: 	Return the Structure "ST_EVENT", it contains the actual 
					event of the Object *)
PROPERTY P_Event : GenLib.ST_EVENT
GET
END_GET
SET
END_SET
END_PROPERTY

{warning 'Eigenschaftenimplementierung hinzufügen'}
(*=== Property: P_FullObjectPath  ============================================

 @param [set]: 	Set the Object Path (Clear String of Object)
 @param [get]: 	Return the Objectpath *)
PROPERTY P_FullObjectPath : STRING
GET
END_GET
SET
END_SET
END_PROPERTY

{warning 'Eigenschaftenimplementierung hinzufügen'}
(*=== Property: P_Global_Ack  ============================================

 @param [set]: 	Set the Bit for Ack from another Object
 @param [get]: 	Return the state of Ack Bit*)
PROPERTY P_Global_Ack : BOOL
GET
END_GET
SET
END_SET
END_PROPERTY

{warning 'Eigenschaftenimplementierung hinzufügen'}
(*=== Property: P_GlobalID  ============================================

 @param [set]: 	-
 @param [get]: 	Return the string of instance path*)
PROPERTY P_GlobalID : STRING
GET
END_GET
END_PROPERTY

END_FUNCTION_BLOCK

// ---- MODULE/SAFETY/POU/FB_ESTOP.TcPOU
FUNCTION_BLOCK FB_ESTOP IMPLEMENTS I_ESTOP
VAR_INPUT
END_VAR
VAR_OUTPUT
END_VAR
VAR //General
	{attribute 'instance-path'} 
    {attribute 'noinit'} 
	strInstancePath:										STRING;
	strFullObjectPath: 										STRING;
	stEvent: 												ST_EVENT;
	bAck: 													BOOL;
	quitDelayTimer:											TON;

	//Interfaces
	itfOpMode:												I_OP_MODE;
	itfQuitEStop:											I_BINARY_OUTPUT;
	itfEStopLoadingLeftState:								I_BINARY_SWITCH;
	itfEStopLoadingRightState: 								I_BINARY_SWITCH;	
	itfEStopWeighSideState:									I_BINARY_SWITCH;
 
	//Schrittkettensteuerung
	eSeq, eLastSeq, eNextSeq:								E_STEP_STATE_ESTOP:=	E_STEP_STATE_ESTOP.ESTOP_PRESSED;
	tonDelay, tonTimeOut, tonStepTime:						TON;
	tDelay:													TIME := T#100MS;
	tTimeOut:												TIME := T#100MS;
	tTimeOutExt:											TIME := T#100MS;
	bDelayActive, bTimeOutActiveQuit, bTimeOutActiveNoQuit:	BOOL;//Timer Option
	bActiveStep, bDebugAcitve, bDebugNext:					BOOL;//Debug Option
	i:														INT;
    iError:													INT; //ERROR-CODE                    	                   		
	listLastSteps:											ARRAY[0..49] OF ST_LAST_STEPS;	
	strExtraInfo:											STRING; 
	eStep_Type:												E_STEP_STATE_TYPE; 
	bDebugModeActive:										BOOL;   
	bWaitForBreakpoint:										BOOL;
	bBreakpointActive:										BOOL;
	bDebugResume:											BOOL;   
	listBreakpoint:											ARRAY[0..10] OF  INT;  
END_VAR

eLastSeq:=eSeq;

CASE eSeq OF 
E_STEP_STATE_ESTOP.BASE:;
		eSeq:=E_STEP_STATE_ESTOP.ESTOP_OK;
	
E_STEP_STATE_ESTOP.RESET:;
		eSeq:=E_STEP_STATE_ESTOP.BASE;

E_STEP_STATE_ESTOP.ESTOP_OK:;
	IF FALSE
		OR itfEStopLoadingLeftState.P_Active
		OR itfEStopLoadingRightState.P_Active
		OR itfEStopWeighSideState.P_Active
	THEN
		eSeq:=E_STEP_STATE_ESTOP.ESTOP_PRESSED;
	ELSE
		itfOpMode.P_EMERGANCY_STOP:=FALSE;
		eSeq:=E_STEP_STATE_ESTOP.ESTOP_OK;
	END_IF

E_STEP_STATE_ESTOP.ESTOP_PRESSED:;
	IF FALSE
		OR itfEStopLoadingLeftState.P_Active
		OR itfEStopLoadingRightState.P_Active
		OR itfEStopWeighSideState.P_Active
	THEN
		itfOpMode.P_EMERGANCY_STOP:=TRUE;
		eSeq:=E_STEP_STATE_ESTOP.ESTOP_PRESSED;
	ELSE
		eSeq:=E_STEP_STATE_ESTOP.WAIT_QUIT_ESTOP;
	END_IF
					
E_STEP_STATE_ESTOP.WAIT_QUIT_ESTOP:;
	IF itfQuitEStop.P_State THEN
		itfQuitEStop.M_Reset();
	END_IF
	IF FALSE
		OR itfEStopLoadingLeftState.P_Active
		OR itfEStopLoadingRightState.P_Active
		OR itfEStopWeighSideState.P_Active
	THEN
		eSeq:=E_STEP_STATE_ESTOP.ESTOP_PRESSED;
	END_IF

E_STEP_STATE_ESTOP.SET_QUIT_ESTOP:;
	itfQuitEStop.M_Set();
	eSeq:=E_STEP_STATE_ESTOP.RESET_QUIT_ESTOP;
	
E_STEP_STATE_ESTOP.RESET_QUIT_ESTOP:;
	quitDelayTimer(IN:= NOT quitDelayTimer.Q, PT := T#500MS);
	IF quitDelayTimer.Q THEN
  		itfQuitEStop.M_Reset();
		eSeq:=E_STEP_STATE_ESTOP.ESTOP_QUIT_OK;
	END_IF
					
E_STEP_STATE_ESTOP.ESTOP_QUIT_OK:;
	eSeq:=E_STEP_STATE_ESTOP.BASE;

(*E_STEP_STATE_ESTOP.TIME_OUT_TO_QUIT:;

	stEvent.bEventActive:=TRUE;
	stEvent.enumEventType:=ENUM_EVENT_TYPE.Rd6_Warning;
	stEvent.strEventText:=concat('Timeout: ',listLastSteps[1].strStepName);
	stEvent.strEventText:=concat(stEvent.strEventText,' > ');
	stEvent.strEventText:=concat(stEvent.strEventText,TO_STRING(listLastSteps[1].tStepTime));
	stEvent.strObject:=strFullObjectPath;
	//Timeout eine Schrittes
	//ENDE	
	IF THIS^.bAck THEN
		eSeq:=eLastSeq;
		stEvent.bEventActive:=FALSE;
	END_IF
E_STEP_STATE_ESTOP.TIME_OUT:;

	stEvent.bEventActive:=TRUE;
	stEvent.enumEventType:=ENUM_EVENT_TYPE.Rd6_Warning;
	stEvent.strEventText:=concat('Timeout: ',listLastSteps[1].strStepName);
	stEvent.strEventText:=concat(stEvent.strEventText,' > ');
	stEvent.strEventText:=concat(stEvent.strEventText,TO_STRING(listLastSteps[1].tStepTime));
	stEvent.strObject:=strFullObjectPath;
	//Timeout eine Schrittes
	//ENDE	

	
E_STEP_STATE_ESTOP.ERROR:;
	
E_STEP_STATE_ESTOP.ERROR_TO_QUIT:;

E_STEP_STATE_ESTOP.ERROR_RESTART:;


E_STEP_STATE_ESTOP.IBN_DUMMY:;
	bDelayActive:=TRUE;
	tDelay:=T#5S;
	IF tonDelay.Q THEN
		eSeq:=E_STEP_STATE_ESTOP.RESET;
	END_IF
	
E_STEP_STATE_ESTOP.DEBUG_BREAK:;
//Warten auf Debug-Bit
IF bDebugNext THEN
	eSeq:=eNextSeq;
	bDebugNext:=FALSE;
END_IF
//Debug Step Ende

ELSE
	eSeq:=E_STEP_STATE_ESTOP.ERROR;
	//ENDE
	
	*)
END_CASE








THIS^._m_SequenceManager();

METHOD PRIVATE _m_DebugManager
VAR_INPUT
	iStepID: int;
END_VAR
IF TRUE
AND THIS^.bDebugModeActive 
AND NOT THIS^.bActiveStep
THEN

THIS^.bBreakpointActive:=TRUE;

FOR i:=0 TO 10 DO
	
	IF TRUE
	AND iStepID=THIS^.listBreakpoint[i] 
	AND iStepID<>0
	THEN
		EXIT;
	END_IF
END_FOR
IF (i<=10) THEN
	THIS^.bBreakpointActive:=TRUE;
END_IF

END_IF
END_METHOD

METHOD _m_Delay : BOOL
VAR_INPUT
	DelayTime:	TIME;
END_VAR
THIS^.bDelayActive:=TRUE;
THIS^.tDelay:=DelayTime;
_m_Delay:=FALSE;
IF THIS^.tonDelay.Q THEN
	_m_Delay:=TRUE;
END_IF
END_METHOD

METHOD PRIVATE _m_GeneralStepSetting : BOOL
VAR_INPUT
	StepType:			E_STEP_STATE_TYPE;
	TimeOutOptions:		E_STEP_STATE_TIMEOUT_OPTION;
	TimeOut:			TIME;
	InfoText:			STRING(20);
	EnableDebug:		BOOL;
	
END_VAR
IF NOT THIS^.bActiveStep THEN

CASE TimeOutOptions OF
	E_STEP_STATE_TIMEOUT_OPTION.NO_TIME_OUT:
		THIS^.bTimeOutActiveNoQuit:=FALSE;
		THIS^.bTimeOutActiveQuit:=FALSE;
		tTimeOut:=T#0S;
	E_STEP_STATE_TIMEOUT_OPTION.TIME_OUT_TO_ERROR:
		THIS^.bTimeOutActiveNoQuit:=TRUE;
		THIS^.bTimeOutActiveQuit:=FALSE;
		tTimeOut:=TimeOut;
	E_STEP_STATE_TIMEOUT_OPTION.TIME_OUT_TO_QUIT:
		THIS^.bTimeOutActiveNoQuit:=FALSE;
		THIS^.bTimeOutActiveQuit:=TRUE;	
		tTimeOut:=TimeOut;
	E_STEP_STATE_TIMEOUT_OPTION.TIME_OUT_TO_RESET:
		THIS^.bTimeOutActiveNoQuit:=TRUE;
		THIS^.bTimeOutActiveQuit:=TRUE;	
		tTimeOut:=TimeOut;
	ELSE
		THIS^.bTimeOutActiveNoQuit:=FALSE;
		THIS^.bTimeOutActiveQuit:=FALSE;
		tTimeOut:=T#0S;;		
END_CASE

THIS^.eStep_Type:=StepType;
THIS^.strExtraInfo:=InfoText;

END_IF
END_METHOD

METHOD PRIVATE _m_SaveLastStep : BOOL
VAR_INPUT
END_VAR
VAR
	i: dint;
END_VAR
IF NOT THIS^.bActiveStep THEN
	
	FOR i:=49 TO 1 BY -1 DO
			listLastSteps[i].strStepName:=listLastSteps[i-1].strStepName;
			listLastSteps[i].tStepTime:=listLastSteps[i-1].tStepTime;
			listLastSteps[i].tDelayTime:=listLastSteps[i-1].tDelayTime;
	END_FOR
	listLastSteps[0].strStepName:=TO_STRING(THIS^.eSeq);
	listLastSteps[1].tStepTime:=THIS^.tonStepTime.ET;
	listLastSteps[1].tStepTime:=THIS^.tonDelay.ET;
ELSE
	listLastSteps[0].tStepTime:=THIS^.tonStepTime.ET;
	listLastSteps[0].tStepTime:=THIS^.tonDelay.ET;	
END_IF
END_METHOD

METHOD PRIVATE _m_SequenceManager
VAR_INPUT
END_VAR


//DelayTimer und TimeOut Timer verwalten
bActiveStep:=eLastSeq=eSeq;
IF NOT bActiveStep THEN
	bDelayActive:=FALSE;
	bTimeOutActiveQuit:=FALSE;
	bTimeOutActiveNoQuit:=FALSE;
END_IF
_m_SaveLastStep();
tonDelay	(IN:=bActiveStep AND bDelayActive, 		PT:=tDelay);
tonTimeOut	(IN:=bActiveStep AND (bTimeOutActiveNoQuit OR bTimeOutActiveQuit), 	PT:=tTimeOut);
tonStepTime	(IN:= bActiveStep, PT:= T#1H);

IF tonTimeOut.Q AND FALSE THEN
	eSeq:=E_STEP_STATE_ESTOP.TIME_OUT;
END_IF

IF iError<>0 THEN
	eSeq:=E_STEP_STATE_ESTOP.ERROR;
END_IF
END_METHOD

METHOD FB_init : BOOL
VAR_INPUT
	bInitRetains : 											BOOL; // if TRUE, the retain variables are initialized (warm start / cold start)
	bInCopyCode : 											BOOL;  // if TRUE, the instance afterwards gets moved into the copy code (online change)
	                                						
    itfOpMode:												I_OP_MODE;
	itfQuitEStop:											I_BINARY_OUTPUT;
	itfEStopLoadingLeftState:								I_BINARY_SWITCH;
	itfEStopLoadingRightState: 								I_BINARY_SWITCH;	
	itfEStopWeighSideState:									I_BINARY_SWITCH;
END_VAR
THIS^.itfOpMode:=						itfOpMode;
THIS^.itfQuitEStop:=					itfQuitEStop;
THIS^.itfEStopLoadingLeftState:=		itfEStopLoadingLeftState;	
THIS^.itfEStopLoadingRightState:= 	    itfEStopLoadingRightState; 	
THIS^.itfEStopWeighSideState:=		    itfEStopWeighSideState;
END_METHOD

METHOD M_Quit : BOOL
VAR_INPUT
END_VAR
IF eSeq=E_STEP_STATE_ESTOP.WAIT_QUIT_ESTOP THEN
	eSeq:=E_STEP_STATE_ESTOP.SET_QUIT_ESTOP;
END_IF
END_METHOD

METHOD M_Reset : BOOL
END_METHOD

(*=== Method: M_Run  ============================================

 @brief: Here is the global code (Timer, Event, Flange,...)*)
METHOD M_Run
END_METHOD

PROPERTY P_E_StopAktiv : BOOL
GET
IF eSeq=E_STEP_STATE_ESTOP.ESTOP_PRESSED THEN
	P_E_StopAktiv:=TRUE;
ELSE
	P_E_StopAktiv:=FALSE;
END_IF
END_GET
END_PROPERTY

PROPERTY P_E_StopLoadingLeftAktiv : BOOL
GET
P_E_StopLoadingLeftAktiv:=NOT THIS^.itfEStopLoadingLeftState.P_Active;
END_GET
END_PROPERTY

PROPERTY P_E_StopLoadingRightAktiv : BOOL
GET
P_E_StopLoadingRightAktiv:=NOT THIS^.itfEStopLoadingRightState.P_Active;
END_GET
END_PROPERTY

PROPERTY P_E_StopQuittieren : BOOL
GET
IF eSeq=E_STEP_STATE_ESTOP.SET_QUIT_ESTOP THEN
	P_E_StopQuittieren:=TRUE;
ELSE
	P_E_StopQuittieren:=FALSE;
END_IF
END_GET
END_PROPERTY

PROPERTY P_E_StopWeighSideAktiv : BOOL
GET
P_E_StopWeighSideAktiv:=NOT THIS^.itfEStopWeighSideState.P_Active;
END_GET
END_PROPERTY

PROPERTY P_ErrorCode : UINT
GET
END_GET
END_PROPERTY

(*=== Property: P_Event  ============================================

 @param [set]: 	Set the Structure "ST_EVENT" from another Object
 @param [get]: 	Return the Structure "ST_EVENT", it contains the actual 
					event of the Object *)
PROPERTY P_Event : GenLib.ST_EVENT
GET
P_Event:=stEvent;
END_GET
SET
stEvent:=P_Event;
END_SET
END_PROPERTY

(*=== Property: P_FullObjectPath  ============================================

 @param [set]: 	Set the Object Path (Clear String of Object)
 @param [get]: 	Return the Objectpath *)
PROPERTY P_FullObjectPath : STRING
GET
P_FullObjectPath:= THIS^.strFullObjectPath;
END_GET
SET
THIS^.strFullObjectPath:=P_FullObjectPath;
END_SET
END_PROPERTY

(*=== Property: P_Global_Ack  ============================================

 @param [set]: 	Set the Bit for Ack from another Object
 @param [get]: 	Return the state of Ack Bit*)
PROPERTY P_Global_Ack : BOOL
GET
P_Global_Ack:=THIS^.bAck;
END_GET
SET
THIS^.bAck:=P_Global_Ack;
END_SET
END_PROPERTY

(*=== Property: P_GlobalID  ============================================

 @param [set]: 	-
 @param [get]: 	Return the string of instance path*)
PROPERTY P_GlobalID : STRING
GET
P_GlobalID:= THIS^.strInstancePath;
END_GET
END_PROPERTY

END_FUNCTION_BLOCK

// ---- MODULE/SAFETY/VISU/FB_VISU_GATE_LOCK.TcPOU
FUNCTION_BLOCK PUBLIC FB_VISU_GATE_LOCK
VAR_INPUT
END_VAR
VAR_OUTPUT
END_VAR
VAR
	itfOpMode:												I_OP_MODE;
	itfUser:												I_USER_MANAGER;
	bClickGateLock:											BOOL;
	itfGateLock:											I_GATE_LOCK;	
	
	bEnable:												BOOL;
	bAdmin:													BOOL;
	sObjName:												STRING;
END_VAR

//Tastensperre bei Auto oder Keiner Betriebsartenauswahl
IF THIS^.itfOpMode.P_OP_MODE_STATE=OP_MODE.MANUAL THEN
	bEnable:=TRUE;
ELSE
	bEnable:=FALSE;
END_IF

bAdmin:=FALSE;
IF itfUser.P_UserGroupID=USER.Admin THEN
	bAdmin:=TRUE;
END_IF

METHOD FB_init : BOOL
VAR_INPUT
	bInitRetains : BOOL; // if TRUE, the retain variables are initialized (warm start / cold start)
	bInCopyCode : BOOL;  // if TRUE, the instance afterwards gets moved into the copy code (online change)
	itfOpMode:												I_OP_MODE;
	itfUser:												I_USER_MANAGER;
	itfDoorLock:											I_GATE_LOCK;
END_VAR
END_METHOD

END_FUNCTION_BLOCK

// ---- IMPLICIT_CHECKS/CheckBounds.TcPOU
// Automatisch erzeugter Code: NICHT EDITIEREN
FUNCTION CheckBounds : DINT
VAR_INPUT
	index, lower, upper: DINT;
END_VAR

// Automatisch erzeugter Code: Es handelt sich hierbei um einen Implementierungsvorschlag.
{noflow}
IF  index < lower THEN
	CheckBounds := lower;
ELSIF  index > upper THEN
	CheckBounds := upper;
ELSE  
	CheckBounds := index;
END_IF
{flow}

END_FUNCTION

// ---- IMPLICIT_CHECKS/CheckDivDInt.TcPOU
// Automatisch erzeugter Code: NICHT EDITIEREN
FUNCTION CheckDivDInt : DINT
VAR_INPUT
	divisor:DINT;
END_VAR

// Automatisch erzeugter Code: Es handelt sich hierbei um einen Implementierungsvorschlag.
{noflow}
IF divisor = 0 THEN
	CheckDivDInt:=1;
ELSE
	CheckDivDInt:=divisor;
END_IF;
{flow}

END_FUNCTION

// ---- IMPLICIT_CHECKS/CheckDivLInt.TcPOU
// Automatisch erzeugter Code: NICHT EDITIEREN
FUNCTION CheckDivLInt : LINT
VAR_INPUT
	divisor:LINT;
END_VAR

// Automatisch erzeugter Code: Es handelt sich hierbei um einen Implementierungsvorschlag.
{noflow}
IF divisor = 0 THEN
	CheckDivLInt:=1;
ELSE
	CheckDivLInt:=divisor;
END_IF;
{flow}

END_FUNCTION

// ---- IMPLICIT_CHECKS/CheckDivLReal.TcPOU
// Automatisch erzeugter Code: NICHT EDITIEREN
FUNCTION CheckDivLReal : LREAL
VAR_INPUT
	divisor:LREAL;
END_VAR

// Automatisch erzeugter Code: Es handelt sich hierbei um einen Implementierungsvorschlag.
{noflow}
IF divisor = 0 THEN
	CheckDivLReal:=1;
ELSE
	CheckDivLReal:=divisor;
END_IF;
{flow}

END_FUNCTION

// ---- IMPLICIT_CHECKS/CheckDivReal.TcPOU
// Automatisch erzeugter Code: NICHT EDITIEREN
FUNCTION CheckDivReal : REAL
VAR_INPUT
	divisor:REAL;
END_VAR

// Automatisch erzeugter Code: Es handelt sich hierbei um einen Implementierungsvorschlag.
{noflow}
IF divisor = 0 THEN
	CheckDivReal:=1;
ELSE
	CheckDivReal:=divisor;
END_IF;
{flow}

END_FUNCTION

// ---- IMPLICIT_CHECKS/CheckLRangeSigned.TcPOU
// Automatisch erzeugter Code: NICHT EDITIEREN
FUNCTION CheckLRangeSigned : LINT
VAR_INPUT
	value, lower, upper: LINT;
END_VAR

// Automatisch erzeugter Code: Es handelt sich hierbei um einen Implementierungsvorschlag.
{noflow}
IF (value < lower) THEN
	CheckLRangeSigned := lower;
ELSIF(value > upper) THEN
	CheckLRangeSigned := upper;
ELSE
	CheckLRangeSigned := value;
END_IF

{flow}

END_FUNCTION

// ---- IMPLICIT_CHECKS/CheckLRangeUnsigned.TcPOU
// Automatisch erzeugter Code: NICHT EDITIEREN
FUNCTION CheckLRangeUnsigned : ULINT
VAR_INPUT
	value, lower, upper: ULINT;
END_VAR

// Automatisch erzeugter Code: Es handelt sich hierbei um einen Implementierungsvorschlag.
{noflow}
IF (value < lower) THEN
	CheckLRangeUnsigned := lower;
ELSIF(value > upper) THEN
	CheckLRangeUnsigned := upper;
ELSE
	CheckLRangeUnsigned := value;
END_IF
{flow}

END_FUNCTION

// ---- IMPLICIT_CHECKS/CheckPointer.TcPOU
// Automatisch erzeugter Code: NICHT EDITIEREN
FUNCTION CheckPointer : POINTER TO BYTE
VAR_INPUT 
	ptToTest : POINTER TO BYTE; // Zieladresse des Pointers
	iSize : DINT;		        // Grösse des Typs auf den der Pointer zeigt. (z.B.: 20 für POINTER TO ARRAY [0..9] OF INT) 
	iGran : DINT;		        // Granularität des Pointer-Zugriffs. Dies ist die Größe des größten nichtstrukturierten Datentyps in dem Typ auf den der Pointer zeigt. (z.B.: 2 für POINTER TO ARRAY [0..9] OF INT)
	bWrite: BOOL;		        // Zeigt Lese- oder Schreibzugriff an. TRUE = Schreibzugriff.
END_VAR

// Automatisch erzeugter Code: Es handelt sich hierbei um einen Implementierungsvorschlag.
{noflow}
IF ptToTest=0 THEN
    ADSLOGSTR(ADSLOG_MSGTYPE_ERROR OR ADSLOG_MSGTYPE_STRING,'CheckPointer failed due to invalid address.','');
ELSIF iSize<=0 THEN
    ADSLOGSTR(ADSLOG_MSGTYPE_ERROR OR ADSLOG_MSGTYPE_STRING,'CheckPointer failed due to invalid size.','');
ELSIF iGran<=0 THEN
    ADSLOGSTR(ADSLOG_MSGTYPE_ERROR OR ADSLOG_MSGTYPE_STRING,'CheckPointer failed due to invalid granularity.','');
// -> Please note that the following memory area check is time consuming:
//ELSIF F_CheckMemoryArea(pData:=ptToTest,nSize:=DINT_TO_UDINT(iSize)) = E_TcMemoryArea.Unknown THEN
//    ADSLOGSTR(ADSLOG_MSGTYPE_ERROR OR ADSLOG_MSGTYPE_STRING,'CheckPointer failed due to unknown memory area.','');
END_IF
CheckPointer := ptToTest;
{flow}

END_FUNCTION

// ---- IMPLICIT_CHECKS/CheckRangeSigned.TcPOU
// Automatisch erzeugter Code: NICHT EDITIEREN
FUNCTION CheckRangeSigned : DINT
VAR_INPUT
	value, lower, upper: DINT;
END_VAR

// Automatisch erzeugter Code: Es handelt sich hierbei um einen Implementierungsvorschlag.
{noflow}
IF (value < lower) THEN
	CheckRangeSigned := lower;
ELSIF(value > upper) THEN
	CheckRangeSigned := upper;
ELSE
	CheckRangeSigned := value;
END_IF
{flow}

END_FUNCTION

// ---- IMPLICIT_CHECKS/CheckRangeUnsigned.TcPOU
// Automatisch erzeugter Code: NICHT EDITIEREN
FUNCTION CheckRangeUnsigned : UDINT
VAR_INPUT
	value, lower, upper: UDINT;
END_VAR

// Automatisch erzeugter Code: Es handelt sich hierbei um einen Implementierungsvorschlag.
{noflow}
IF (value < lower) THEN
	CheckRangeUnsigned := lower;
ELSIF(value > upper) THEN
	CheckRangeUnsigned := upper;
ELSE
	CheckRangeUnsigned := value;
END_IF
{flow}

END_FUNCTION

// ---- ORGANISATION/GENERAL/ITF/FB_Abstract_FunktionCtrl.TcPOU
FUNCTION_BLOCK ABSTRACT FB_Abstract_FunktionCtrl IMPLEMENTS I_FunctionCtrl
VAR_INPUT
END_VAR
VAR_OUTPUT
END_VAR
VAR
END_VAR

{warning 'Eigenschaftenimplementierung hinzufügen'}
PROPERTY Busy : BOOL
GET
END_GET
END_PROPERTY

{warning 'Eigenschaftenimplementierung hinzufügen'}
PROPERTY Done : BOOL
GET
END_GET
END_PROPERTY

{warning 'Eigenschaftenimplementierung hinzufügen'}
PROPERTY Error : BOOL
GET
END_GET
END_PROPERTY

{warning 'Eigenschaftenimplementierung hinzufügen'}
PROPERTY ErrorCode : WORD
GET
END_GET
END_PROPERTY

{warning 'Methodenimplementierung hinzufügen'}
METHOD Execute : BOOL
END_METHOD

{warning 'Eigenschaftenimplementierung hinzufügen'}
PROPERTY Ready : BOOL
GET
END_GET
END_PROPERTY

{warning 'Methodenimplementierung hinzufügen'}
METHOD Reset : BOOL
END_METHOD

END_FUNCTION_BLOCK

// ---- ORGANISATION/GENERAL/POU/FB_GENERAL.TcPOU
{attribute 'reflection'} 
FUNCTION_BLOCK ABSTRACT FB_GENERAL
VAR //General
  	{attribute 'instance-path'} 
    {attribute 'noinit'} 
	strInstancePath: 	STRING;
END_VAR

METHOD M_CyclicRun : BOOL
VAR_INPUT
END_VAR
END_METHOD

PROPERTY P_ObjectID : STRING
GET
P_ObjectID:='dfknhkljsfa';
END_GET
SET
END_SET
END_PROPERTY

END_FUNCTION_BLOCK

// ---- ORGANISATION/OP_MODE/POU/FB_OP_MODE.TcPOU
FUNCTION_BLOCK FB_OP_MODE IMPLEMENTS I_OP_MODE

VAR
	bAutomatic						: BOOL;
	bDebug							: BOOL;
	bManual							: BOOL;
	bReset							: BOOL;
	btemporay_Automatic				: BOOL;
	btemporay_Debug					: BOOL;
	btemporay_Manual				: BOOL;
	btemporay_Reset					: BOOL;
	bInitOK							: BOOL;
	bMachineStateOK					: BOOL;
	bControlOn						: BOOL;
	bEmergancyStop					: BOOL;
	bFatalError						: BOOL;
	itfHandleEvents					: I_HANDLE_EVENTS;
	itfControlOn					: I_BINARY_SWITCH;
	itfControlIsOn					: I_BINARY_OUTPUT;
	itfMainAirOk					: I_BINARY_SWITCH;
END_VAR


//Check the Machine State
bMachineStateOK:= TRUE;
bControlOn:= TRUE;
IF NOT itfControlOn.P_Active OR NOT itfMainAirOk.P_Active 
OR P_EMERGANCY_STOP
OR itfHandleEvents.P_State >= ENUM_EVENT_TYPE.Rd6_Warning THEN
	bMachineStateOK:= FALSE;
	bControlOn:= FALSE;
	M_OP_MODE_OFF();		
END_IF

IF bControlOn THEN
	itfControlIsOn.M_Set();
ELSE
	itfControlIsOn.M_Reset();
END_IF

METHOD FB_init : BOOL
VAR_INPUT
	bInitRetains : BOOL; // if TRUE, the retain variables are initialized (warm start / cold start)
	bInCopyCode : BOOL;  // if TRUE, the instance afterwards gets moved into the copy code (online change)
	itfHandleEvents: I_HANDLE_EVENTS;
	//itfControlOn: I_BINARY_SWITCH;
	//itfControlIsOn: I_BINARY_OUTPUT;
	//itfMainAirOk:  I_BINARY_SWITCH;
END_VAR
THIS^.itfHandleEvents:=itfHandleEvents;
//THIS^.itfControlOn:= itfControlOn;
//THIS^.itfControlIsOn:= itfControlIsOn;
//THIS^.itfMainAirOk:= itfMainAirOk;
END_METHOD

METHOD M_AUTOMATIC
IF NOT bAutomatic 
	(*AND NOT bDebug 
	AND NOT bManual 
	AND NOT bReset*) THEN
		//set Temporary OP Mode
		IF NOT btemporay_Automatic THEN
			btemporay_Automatic	:= TRUE;
			btemporay_Debug		:= FALSE;
			btemporay_Manual	:= FALSE;
			btemporay_Reset		:= FALSE;
		ELSE
			btemporay_Automatic	:= FALSE;
			btemporay_Debug		:= FALSE;
			btemporay_Manual	:= FALSE;
			btemporay_Reset		:= FALSE;	
		END_IF
END_IF;
END_METHOD

METHOD M_DEBUG
IF (*NOT bAutomatic 
	AND*) NOT bDebug 
	(*AND NOT bManual 
	AND NOT bReset*) THEN
		//set Temporary OP Mode
		IF NOT btemporay_Debug THEN
			btemporay_Automatic	:= FALSE;
			btemporay_Debug		:= TRUE;
			btemporay_Manual	:= FALSE;
			btemporay_Reset		:= FALSE;
		ELSE
			btemporay_Automatic	:= FALSE;
			btemporay_Debug		:= FALSE;
			btemporay_Manual	:= FALSE;
			btemporay_Reset		:= FALSE;
		END_IF
END_IF;
END_METHOD

METHOD M_MANUAL
IF (*NOT bAutomatic 
	AND NOT bDebug 
	AND*) NOT bManual 
	(*AND NOT bReset*) THEN
		//set Temporary OP Mode
		IF NOT btemporay_Manual THEN
			btemporay_Automatic	:= FALSE;
			btemporay_Debug		:= FALSE;
			btemporay_Manual	:= TRUE;
			btemporay_Reset		:= FALSE;
		ELSE
			btemporay_Automatic	:= FALSE;
			btemporay_Debug		:= FALSE;
			btemporay_Manual	:= FALSE;
			btemporay_Reset		:= FALSE;	
		END_IF
END_IF;
END_METHOD

METHOD M_OP_MODE_OFF
//every OP Mode off
bAutomatic	:= FALSE;
bDebug		:= FALSE;
bManual		:= FALSE;
bReset		:= FALSE;
btemporay_Automatic	:= FALSE;
btemporay_Debug		:= FALSE;
btemporay_Manual	:= FALSE;
btemporay_Reset		:= FALSE;
END_METHOD

METHOD M_OP_MODE_ON : BOOL
//Automtic on
IF btemporay_Automatic THEN
	bAutomatic			:= TRUE;
	bDebug				:= FALSE;
	bManual				:= FALSE;
	bReset				:= FALSE;
	btemporay_Automatic := FALSE;
	btemporay_Debug     := FALSE;
	btemporay_Manual    := FALSE;
	btemporay_Reset     := FALSE;
END_IF
//Debug on
IF btemporay_Debug THEN
	bAutomatic			:= FALSE;
	bDebug				:= TRUE;
	bManual				:= FALSE;
	bReset				:= FALSE;
	btemporay_Automatic := FALSE;
	btemporay_Debug     := FALSE;
	btemporay_Manual    := FALSE;
	btemporay_Reset     := FALSE;
END_IF
//Manual on
IF btemporay_Manual THEN
	bAutomatic			:= FALSE;
	bDebug				:= FALSE;
	bManual				:= TRUE;
	bReset				:= FALSE;
	btemporay_Automatic := FALSE;
	btemporay_Debug     := FALSE;
	btemporay_Manual    := FALSE;
	btemporay_Reset     := FALSE;
END_IF
//Reset on
IF btemporay_Reset THEN
	bAutomatic			:= FALSE;
	bDebug				:= FALSE;
	bManual				:= FALSE;
	bReset				:= TRUE;
	btemporay_Automatic := FALSE;
	btemporay_Debug     := FALSE;
	btemporay_Manual    := FALSE;
	btemporay_Reset     := FALSE;
END_IF
END_METHOD

METHOD M_RESET : BOOL
IF (*NOT bAutomatic 
	AND NOT bDebug 
	AND NOT bManual 
	AND*) NOT bReset THEN
		//set Temporary OP Mode
			IF NOT btemporay_Reset THEN
			btemporay_Automatic	:= FALSE;
			btemporay_Debug		:= FALSE;
			btemporay_Manual	:= FALSE;
			btemporay_Reset		:= TRUE;
		ELSE
			btemporay_Automatic	:= FALSE;
			btemporay_Debug		:= FALSE;
			btemporay_Manual	:= FALSE;
			btemporay_Reset		:= FALSE;	
		END_IF
END_IF;
END_METHOD


PROPERTY P_CONTROL_ON : BOOL
GET
P_CONTROL_ON:= bControlOn;
END_GET
SET
bControlOn:= P_CONTROL_ON;
END_SET
END_PROPERTY

PROPERTY P_EMERGANCY_STOP : BOOL
GET
P_EMERGANCY_STOP:= bEmergancyStop;
END_GET
SET
bEmergancyStop:=P_EMERGANCY_STOP;
END_SET
END_PROPERTY

{warning 'Eigenschaftenimplementierung hinzufügen'}
PROPERTY P_INIT_OK : BOOL
GET
P_INIT_OK := THIS^.P_OP_MODE_STATE = OP_MODE.INIT_OK;
END_GET
SET
THIS^.bInitOK := P_INIT_OK;
END_SET
END_PROPERTY

PROPERTY P_OP_MODE_STATE : INT
GET
VAR
	thne: INT;
END_VAR
//MACHINE STATE
IF P_CONTROL_ON AND THIS^.itfMainAirOk.P_Active THEN
	P_OP_MODE_STATE:=OP_MODE.MAIN_AIR_OK;
END_IF

IF P_CONTROL_ON THEN
	P_OP_MODE_STATE:=OP_MODE.CONTROL_ON;
END_IF

IF itfHandleEvents.P_State > ENUM_EVENT_TYPE.Rd6_Warning THEN
	P_OP_MODE_STATE:=OP_MODE.MACHINE_ERROR;
END_IF

IF P_EMERGANCY_STOP THEN
	P_OP_MODE_STATE:=OP_MODE.SAFETY_STOP;
END_IF





//OP MODE

IF bAutomatic AND bMachineStateOK 	THEN
	P_OP_MODE_STATE:=OP_MODE.AUTO;
END_IF;
			
IF bDebug AND bMachineStateOK 		THEN
	P_OP_MODE_STATE:=OP_MODE.DEBUG;
END_IF

IF bManual	AND bMachineStateOK 	THEN
	P_OP_MODE_STATE:=OP_MODE.MANUAL;
END_IF

IF  bReset	AND bMachineStateOK 	THEN
	P_OP_MODE_STATE:=OP_MODE.INIT;
END_IF

IF bInitOK AND bMachineStateOK THEN
	P_OP_MODE_STATE:=OP_MODE.INIT_OK;
END_IF

//OP MODE TEMP

IF btemporay_Automatic	AND bMachineStateOK THEN
	P_OP_MODE_STATE:=OP_MODE.AUTO_TEMPORARY;
END_IF

IF btemporay_Debug AND bMachineStateOK 	THEN
	P_OP_MODE_STATE:=OP_MODE.DEBUG_TEMPORARY;
END_IF

IF btemporay_Manual	AND bMachineStateOK THEN
	P_OP_MODE_STATE:=OP_MODE.MANUAL_TEMPORARY;
END_IF

IF btemporay_Reset AND bMachineStateOK 	THEN
	P_OP_MODE_STATE:=OP_MODE.RESET_TEMPORARY;
END_IF
END_GET
END_PROPERTY

{warning 'Eigenschaftenimplementierung hinzufügen'}
PROPERTY P_QUIT : BOOL
GET
END_GET
END_PROPERTY

END_FUNCTION_BLOCK

// ---- ORGANISATION/OP_MODE/POU/FB_OP_MODE_HMI.TcPOU
FUNCTION_BLOCK FB_OP_MODE_HMI
VAR
	itfOpMode:  I_OP_MODE;
	
//Press 
	bClick_Reset					: BOOL;
	bClick_Start					: BOOL;
	bClick_Stop						: BOOL;
	bClickPause						: BOOL;
	

//State
	bStateStart						: BOOL;
	bStateStop						: BOOL;
	bStatePause						: BOOL;
	bStateReset						: BOOL;
	

//Enable
	bEnableStart					: BOOL:=TRUE;
	bEnableStop						: BOOL:=TRUE;
	bEnablePause					: BOOL:=TRUE;
	bEnableReset					: BOOL:=TRUE;
	
//Options
	bEnableCalibration				: BOOL;
	bOptionCalibration				: BOOL;
	
	bEnableStepByStep				: BOOL;
	bOptionStepByStep				: BOOL;
	
	bEnableEmptyRun					: BOOL;
	bOptionEmptyRun					: BOOL;
	
	
//TextlistID
	nTexlistID						: INT;
	
	fbBlink							: FB_Blink;
END_VAR
VAR_IN_OUT

END_VAR
VAR
END_VAR

IF bClick_Start THEN
	bClick_Start:=FALSE;
	nTexlistID:=nTexlistID+1;
	IF NOT bStateStart THEN
		bStateStart:=TRUE;
		bStateStop:=FALSE;
		bStatePause:=FALSE;
	ELSE
		bStateStart:=FALSE;
	END_IF
END_IF

IF bClick_Stop THEN
	bClick_Stop:=FALSE;
	nTexlistID:=nTexlistID-1;
	IF NOT bStateStop THEN
		bStateStop:=TRUE;
		bStateStart:=FALSE;
		bStatePause:=FALSE;
	ELSE
		bStateStop:=FALSE;
	END_IF
END_IF

IF bClickPause THEN
	bClickPause:=FALSE;
	nTexlistID:=nTexlistID+1;
	IF NOT bStateStop THEN
		bStatePause:=TRUE;
		bStateStop:=FALSE;
		bStateStart:=FALSE;
	ELSE
		bStatePause:=FALSE;
	END_IF
END_IF

METHOD FB_init : BOOL
VAR_INPUT
	bInitRetains : BOOL; // if TRUE, the retain variables are initialized (warm start / cold start)
	bInCopyCode : BOOL;  // if TRUE, the instance afterwards gets moved into the copy code (online change)
	itfOpMode:  I_OP_MODE;
END_VAR
this^.itfOpMode:= itfOpMode;
END_METHOD

END_FUNCTION_BLOCK

// ---- ORGANISATION/OP_MODE/POU/FB_OP_MODE_VISU.TcPOU
FUNCTION_BLOCK FB_OP_MODE_VISU
VAR
	itfOpMode:  I_OP_MODE;
	//Press 
	bClick_Automatic				: BOOL;
	bClick_Debug					: BOOL;
	bClick_Manual					: BOOL;
	bClick_Reset					: BOOL;
	bClick_Start					: BOOL;
	bClick_Stop						: BOOL;
	bClickPause						: BOOL;
	//State
	b_Automatic						: BOOL;
	b_Debug							: BOOL;
	b_Manual						: BOOL;
	b_Reset							: BOOL;
	//temporay State
	btemporay_Automatic				: BOOL;
	btemporay_Debug					: BOOL;
	btemporay_Manual				: BOOL;
	btemporay_Reset					: BOOL;
	iOPModeState					: INT;
	
	fbBlink							: FB_Blink;
END_VAR
VAR_IN_OUT

END_VAR
VAR
END_VAR


//CLICK to OP-Mode
IF bClick_Automatic		THEN
	itfOpMode.M_AUTOMATIC();
	 bClick_Automatic	:= FALSE;
END_IF
	
IF bClick_Debug			THEN
	itfOpMode.M_DEBUG();
	bClick_Debug		:= FALSE;
END_IF
		
IF bClick_Manual		THEN
	itfOpMode.M_MANUAL();
	bClick_Manual		:= FALSE;
END_IF
			
IF bClick_Reset			THEN
	itfOpMode.M_RESET();
	bClick_Reset		:= FALSE;
END_IF
	
		
IF bClick_Start			THEN
	itfOpMode.M_OP_MODE_ON();
	bClick_Start		:= FALSE;
END_IF
		
IF  bClick_Stop			THEN
	itfOpMode.M_OP_MODE_OFF();
	bClick_Stop			:= FALSE;
END_IF
//
b_Automatic				:= FALSE;
b_Debug					:= FALSE; 
b_Manual				:= FALSE;
b_Reset					:= FALSE;
btemporay_Automatic		:= FALSE;
btemporay_Debug			:= FALSE;
btemporay_Manual		:= FALSE;
btemporay_Reset			:= FALSE;

//GET OP MODE STATE
CASE itfOpMode.P_OP_MODE_STATE OF		
	OP_MODE.AUTO: 				b_Automatic:= TRUE;
 	OP_MODE.DEBUG:				b_Debug:= TRUE;
	OP_MODE.MANUAL:				b_Manual:= TRUE;
	OP_MODE.INIT:				b_Reset:= TRUE;
	OP_MODE.AUTO_TEMPORARY:		btemporay_Automatic:= TRUE;
	OP_MODE.DEBUG_TEMPORARY:	btemporay_Debug:= TRUE;
	OP_MODE.MANUAL_TEMPORARY:	btemporay_Manual:= TRUE;
	OP_MODE.RESET_TEMPORARY:	btemporay_Reset:= TRUE;
	OP_MODE.ACTIVATE_PAUSE: 	btemporay_Automatic:=fbBlink.P_2Hz;
	OP_MODE.IN_PAUSE:			btemporay_Automatic:= TRUE;
END_CASE
iOPModeState:=itfOpMode.P_OP_MODE_STATE;

METHOD FB_init : BOOL
VAR_INPUT
	bInitRetains : BOOL; // if TRUE, the retain variables are initialized (warm start / cold start)
	bInCopyCode : BOOL;  // if TRUE, the instance afterwards gets moved into the copy code (online change)
	itfOpMode:  I_OP_MODE;
END_VAR
this^.itfOpMode:= itfOpMode;
END_METHOD

END_FUNCTION_BLOCK

// ---- ORGANISATION/USER_MANAGER/POU/FB_ESTOP_RESET.TcPOU
FUNCTION_BLOCK FB_ESTOP_RESET
VAR_INPUT
END_VAR
VAR_OUTPUT
END_VAR
VAR
	
END_VAR

END_FUNCTION_BLOCK

// ---- POUs/F_SEND_EVENTLOGGER_MSG.TcPOU
FUNCTION F_SEND_EVENTLOGGER_MSG : BOOL
VAR_INPUT
	fbMessage:									TcEventEntry;
END_VAR
VAR
	bInit : 									BOOL; 
    bSend : 									BOOL; 
    fbMsg : 									FB_TcMessage; 
END_VAR

IF( fbMessage.nEventId = GVL_EventLogger.fbPrevMsg.nEventId
	AND fbMessage.eSeverity = GVL_EventLogger.fbPrevMsg.eSeverity) THEN
	bInit:=FALSE;
	bSend:=FALSE;
ELSE
	bInit:=TRUE;
	bSend:=TRUE;
END_IF

IF bInit THEN
    bInit := FALSE; 
    fbMsg.CreateEx(fbMessage, 0); 
END_IF

IF bSend THEN 
    bSend := FALSE; 
    fbMsg.Send(0); 
	GVL_EventLogger.fbPrevMsg:=fbMessage;
	GVL_EventLogger.udiPrevMsgId:=fbMessage.nEventId;
END_IF

END_FUNCTION

// ---- GlobalTextList.TcGTLO
TEXTLIST GlobalTextList
  1706 = ' '
  2550 = ' Baudrate: %d' | de: ' Baudrate: %d' | en: ' Baudrate: %d'
  2541 = ' Bits/s: %8.0f' | de: ' Bits/s: %8.0f' | en: ' Bits/s: %8.0f'
  467 = ' Busy:     %s' | de: ' Busy:     %s' | en: ' Busy:     %s'
  1579 = ' Bytes:\n %d' | de: ' Bytes:\n %d' | en: ' Bytes:\n %d'
  2203 = ' ca. %3.1f %% of baud rate' | de: ' ca. %3.1f %% of baud rate' | en: ' ca. %3.1f %% of baud rate'
  2186 = ' ComPort: %d' | de: ' ComPort: %d' | en: ' ComPort: %d'
  464 = ' CTS:    %s' | de: ' CTS:    %s' | en: ' CTS:    %s'
  2170 = ' DataBits:  %d' | de: ' DataBits:  %d' | en: ' DataBits:  %d'
  465 = ' DSR:    %s' | de: ' DSR:    %s' | en: ' DSR:    %s'
  462 = ' DTR:    %s' | de: ' DTR:    %s' | en: ' DTR:    %s'
  2570 = ' Error:    %d' | de: ' Error:    %d' | en: ' Error:    %d'
  470 = " NetId: '%s'" | de: " NetId: '%s'" | en: " NetId: '%s'"
  2162 = ' Parity:       %s' | de: ' Parity:       %s' | en: ' Parity:       %s'
  469 = ' PortOpen: %s' | de: ' PortOpen: %s' | en: ' PortOpen: %s'
  2211 = ' RTS:    %s' | de: ' RTS:    %s' | en: ' RTS:    %s'
  2560 = ' SendDelay: %s' | de: ' SendDelay: %s' | en: ' SendDelay: %s'
  2178 = ' StopBits:  %d' | de: ' StopBits:  %d' | en: ' StopBits:  %d'
  1592 = ' SumRcvBytes:   %d' | de: ' SumRcvBytes:   %d' | en: ' SumRcvBytes:   %d'
  2195 = ' SumSentBytes: %d' | de: ' SumSentBytes: %d' | en: ' SumSentBytes: %d'
  2154 = ' TelRcv:   %d' | de: ' TelRcv:   %d' | en: ' TelRcv:   %d'
  2580 = ' TelSent: %d' | de: ' TelSent: %d' | en: ' TelSent: %d'
  475 = ' TraceL.:  %d' | de: ' TraceL.:  %d' | en: ' TraceL.:  %d'
  477 = ' TxData:' | de: ' TxData:' | en: ' TxData:'
  474 = ' TxData[ascii]: %s' | de: ' TxData[ascii]: %s' | en: ' TxData[ascii]: %s'
  472 = ' TxData[hex]:   %s' | de: ' TxData[hex]:   %s' | en: ' TxData[hex]:   %s'
  854 = '%' | de: '%' | en: '%'
  66 = '%.0f' | de: '%.0f' | en: '%.0f'
  991 = '%.2f' | de: '%.2f' | en: '%.2f'
  162 = '%.3f' | de: '%.3f' | en: '%.3f'
  2043 = '%1.2f' | de: '%1.2f' | en: '%1.2f'
  1004 = '%1.3f'
  937 = '%1.4' | de: '%1.4' | en: '%1.4'
  3525 = '%1.4f' | de: '%1.4f' | en: '%1.4f'
  321 = '%2.1' | de: '%2.1' | en: '%2.1'
  468 = '%2.1f' | de: '%2.1f' | en: '%2.1f'
  4586 = '%2.2f'
  305 = '%2.3f' | de: '%2.3f' | en: '%2.3f'
  1978 = '%2.4' | de: '%2.4' | en: '%2.4'
  2988 = '%3.0f' | de: '%3.0f' | en: '%3.0f'
  143 = '%3.1f' | de: '%3.1f' | en: '%3.1f'
  481 = '%3.2f' | de: '%3.2f' | en: '%3.2f'
  3808 = '%3.3f'
  46 = '%3.4f' | de: '%3.4f' | en: '%3.4f'
  2349 = '%4.1' | de: '%4.1' | en: '%4.1'
  3862 = '%4.1f' | de: '%4.1f' | en: '%4.1f'
  3302 = '%5.1f' | de: '%5.1f' | en: '%5.1f'
  1186 = '%5.2f' | de: '%5.2f' | en: '%5.2f'
  3061 = '%5.4f' | de: '%5.4f' | en: '%5.4f'
  3305 = '%5.5f' | de: '%5.5f' | en: '%5.5f'
  1547 = '%5.5f '
  5935 = '%5.5f 1/min'
  4924 = '%5.5f A'
  6836 = '%5.5f kg'
  2191 = '%5.5f mm'
  5001 = '%5.5f mV'
  2223 = '%5.5f N'
  1102 = '%5.5f V'
  5084 = '%5.5f °'
  2878 = '%7.3f' | de: '%7.3f' | en: '%7.3f'
  994 = '%d' | de: '%d' | en: '%d'
  992 = '%f' | de: '%f' | en: '%f'
  3702 = '%f2.3' | de: '%f2.3' | en: '%f2.3'
  1028 = '%i' | de: '%i' | en: '%i'
  844 = '%s' | de: '%s' | en: '%s'
  1762 = "'Override in %'" | de: "'Override in %'" | en: "'Override in %'"
  1609 = '+' | de: '+' | en: '+'
  2200 = '+ +' | de: '+ +' | en: '+ +'
  2422 = '-' | de: '-' | en: '-'
  3000 = '- -' | de: '- -' | en: '- -'
  3443 = '--'
  1288 = '0' | de: '0' | en: '0'
  1306 = '0-10V' | de: '0-10V' | en: '0-10V'
  334 = '1' | de: '1' | en: '1'
  4938 = '1/0'
  3374 = '15Pin'
  676 = '2' | de: '2' | en: '2'
  5713 = '24Pin'
  11 = '3' | de: '3' | en: '3'
  955 = '4' | de: '4' | en: '4'
  754 = '4-20mA' | de: '4-20mA' | en: '4-20mA'
  1273 = '5' | de: '5' | en: '5'
  841 = '6' | de: '6' | en: '6'
  645 = '7' | de: '7' | en: '7'
  1477 = '900;1200;1500;1800;2500;3300'
  2022 = '900;1200;1500;1800;2500;3300;'
  440 = ':= read_input_boolean_register(address)' | de: ':= read_input_boolean_register(address)' | en: ':= read_input_boolean_register(address)'
  999 = ':= read_input_float_register(address)' | de: ':= read_input_float_register(address)' | en: ':= read_input_float_register(address)'
  234 = ':= read_input_integer_register(address)' | de: ':= read_input_integer_register(address)' | en: ':= read_input_integer_register(address)'
  23 = ':= read_output_boolean_register(address)' | de: ':= read_output_boolean_register(address)' | en: ':= read_output_boolean_register(address)'
  80 = ':= read_output_float_register(address)' | de: ':= read_output_float_register(address)' | en: ':= read_output_float_register(address)'
  1213 = ':= read_output_integer_register(address)' | de: ':= read_output_integer_register(address)' | en: ':= read_output_integer_register(address)'
  3344 = ':=1' | de: ':=1' | en: ':=1'
  987 = '< :' | de: '< :' | en: '< :'
  986 = '<= :' | de: '<= :' | en: '<= :'
  985 = '> :' | de: '> :' | en: '> :'
  984 = '>= :' | de: '>= :' | en: '>= :'
  213 = '?' | de: '?' | en: '?'
  1773 = 'ABBRUCH' | de: 'ABBRUCH' | en: 'CANCEL'
  97 = 'Absolut' | de: 'Absolut' | en: 'Absolut'
  660 = 'ABWAHL ALLE' | de: 'ABWAHL ALLE' | en: 'DESELECT ALL'
  5197 = 'Achtung Abstufung im UPV verwenden'
  39 = 'Active' | de: 'Active' | en: 'Active'
  161 = 'Actual Value' | de: 'Actual Value' | en: 'Actual Value'
  2723 = 'Admin' | de: 'Admin' | en: 'Admin'
  612 = 'ADRESS' | de: 'ADRESS' | en: 'ADRESS'
  2919 = 'After' | de: 'After' | en: 'After'
  328 = 'agdfgs' | de: 'agdfgs' | en: 'agdfgs'
  6839 = 'Akivate'
  2832 = 'Aktuelle Position'
  4339 = 'Aktueller Druck'
  2016 = 'Analog'
  217 = 'analog_in[0]' | de: 'analog_in[0]' | en: 'analog_in[0]'
  1145 = 'analog_in[1]' | de: 'analog_in[1]' | en: 'analog_in[1]'
  356 = 'analog_in[2]' | de: 'analog_in[2]' | en: 'analog_in[2]'
  1323 = 'analog_in[3]' | de: 'analog_in[3]' | en: 'analog_in[3]'
  914 = 'analog_out[0]' | de: 'analog_out[0]' | en: 'analog_out[0]'
  1334 = 'analog_out[1]' | de: 'analog_out[1]' | en: 'analog_out[1]'
  848 = 'analog_out[2]' | de: 'analog_out[2]' | en: 'analog_out[2]'
  695 = 'analog_out[3]' | de: 'analog_out[3]' | en: 'analog_out[3]'
  1524 = 'Analysis' | de: 'Analysis' | en: 'Analysis'
  3597 = 'ANGLE (°)' | de: 'ANGLE (°)' | en: 'ANGLE (°)'
  1031 = 'angle of throttle:' | de: 'angle of throttle:' | en: 'angle of throttle:'
  2689 = 'ANGLEl (°)'
  2843 = 'ANWAHL ALLE' | de: 'ANWAHL ALLE' | en: 'SELECT ALL'
  2202 = 'Anzahl Zeichen DMC'
  1699 = 'Anzeigename'
  149 = 'Anzeigetext:' | de: 'Anzeigetext:' | en: 'Ad text:'
  5385 = 'asfasdf'
  4209 = 'Auftragsnummer:\t\t%s'
  1486 = 'Auslastung (%):' | de: 'Auslastung (%):' | en: 'Workload (%):'
  6065 = 'Auswahl Betriebsmodus'
  5171 = 'Auswahl Greifkraft'
  3491 = 'Auswahl Programmnummer:%i'
  4332 = 'Auswahl Sequenz'
  3066 = 'Auswertung Kamera'
  1458 = 'AUTO' | de: 'AUTO' | en: 'AUTO'
  14 = 'Auto Inc.' | de: 'Auto Inc.' | en: 'Auto Inc.'
  166 = 'AUTOMATIC' | de: 'AUTOMATIC' | en: 'AUTOMATIC'
  550 = 'Automatic Retest'
  5108 = 'Automatic Retest7'
  177 = 'Axis' | de: 'Axis' | en: 'Axis'
  867 = 'AXIS TCP' | de: 'AXIS TCP' | en: 'AXIS TCP'
  180 = 'Band' | de: 'Band' | en: 'Band'
  1548 = 'BAND' | de: 'BAND' | en: 'BAND'
  1604 = 'Band 1'
  2562 = 'Band 2'
  4376 = 'Band 3'
  6525 = 'Band 4'
  4099 = 'Band 5'
  241 = 'Band 6'
  5767 = 'Band 7'
  3445 = 'Band 8'
  794 = 'BASE' | de: 'BASE' | en: 'BASE'
  4461 = 'Base'
  482 = 'BCC:\n %' | de: 'BCC:\n %' | en: 'BCC:\n %'
  139 = 'BCC:\n %x' | de: 'BCC:\n %x' | en: 'BCC:\n %x'
  1662 = 'Before' | de: 'Before' | en: 'Before'
  1211 = 'Beladen fertig' | de: 'Beladen fertig' | en: 'Beladen fertig'
  732 = 'Blow' | de: 'Blow' | en: 'Blow'
  476 = 'BLOW' | de: 'BLOW' | en: 'BLOW'
  4341 = 'Bohrung gefunden'
  533 = 'Camline NIO Teil entladen' | de: 'Camline NIO Teil entladen' | en: 'Camline NIO Teil entladen'
  198 = 'CANCEL' | de: 'CANCEL' | en: 'CANCEL'
  1621 = 'Channel 1 Common'
  1558 = 'Checkbox' | de: 'Checkbox' | en: 'Checkbox'
  707 = 'CLOSE' | de: 'CLOSE' | en: 'CLOSE'
  1673 = 'CLOSE DOOR'
  1392 = 'Cobot 1 an M400' | de: 'Cobot 1 an M400' | en: 'Cobot 1 an M400'
  995 = 'Cobot 2 an M400' | de: 'Cobot 2 an M400' | en: 'Cobot 2 an M400'
  1664 = 'Cobot 2 an M500' | de: 'Cobot 2 an M500' | en: 'Cobot 2 an M500'
  1378 = 'Cobot Active' | de: 'Cobot Active' | en: 'Cobot Active'
  1752 = 'Cobot Aktiv' | de: 'Cobot Aktiv' | en: 'Cobot Aktiv'
  1410 = 'Cobot: Beladen' | de: 'Cobot: Beladen' | en: 'Cobot: Beladen'
  839 = 'Cobot: Entladen' | de: 'Cobot: Entladen' | en: 'Cobot: Entladen'
  2531 = 'compare ok' | de: 'compare ok' | en: 'compare ok'
  1567 = 'Compare On' | de: 'Compare On' | en: 'Compare On'
  338 = 'Compl. Current in A:'
  1414 = 'Compl. Current in mA:'
  4747 = 'Complete Test'
  1536 = 'Config' | de: 'Config' | en: 'Config'
  714 = 'Configuratible Inputs' | de: 'Configuratible Inputs' | en: 'Configuratible Inputs'
  1332 = 'Configuratible Outputs' | de: 'Configuratible Outputs' | en: 'Configuratible Outputs'
  16 = 'Connect' | de: 'Connect' | en: 'Connect'
  2757 = 'Const Time' | de: 'Const Time' | en: 'Const Time'
  784 = 'Const. Slope'
  3622 = 'Const. Time'
  3549 = 'Constant-Time'
  479 = 'Continuous Send Mode' | de: 'Continuous Send Mode' | en: 'Continuous Send Mode'
  1573 = 'Continuous Send On' | de: 'Continuous Send On' | en: 'Continuous Send On'
  586 = 'controller major version:' | de: 'controller major version:' | en: 'controller major version:'
  875 = 'controller minor version:' | de: 'controller minor version:' | en: 'controller minor version:'
  1705 = 'CONVOYER' | de: 'CONVOYER' | en: 'CONVOYER'
  1919 = 'Convoyer' | de: 'Convoyer' | en: 'Convoyer'
  119 = 'Cool' | de: 'Cool' | en: 'Cool'
  1804 = 'COPY'
  1620 = 'CREATE' | de: 'CREATE' | en: 'CREATE'
  349 = 'Cur' | de: 'Cur' | en: 'Cur'
  3929 = 'Current 1'
  4560 = 'Current 2'
  28 = 'Current Joint 0:' | de: 'Current Joint 0:' | en: 'Current Joint 0:'
  3535 = 'Current Range: Max.'
  4510 = 'Current Range: Max. in mA:'
  2999 = 'Current Range: Min.'
  4840 = 'Current Range: Min. in mA:'
  553 = 'Daimler' | de: 'Daimler' | en: 'Daimler'
  3334 = 'Daten von MaXYmos'
  2739 = 'Dauertest'
  1327 = 'Delaytime to automatic retest'
  5080 = 'delaytime to next automatic retest'
  529 = 'DELETE' | de: 'DELETE' | en: 'DELETE'
  1540 = 'Delete'
  4644 = 'Delete Parameter Settings?'
  3088 = 'Delete Parameter-Settings?'
  398 = 'DELETE POPUP'
  126 = 'Delta Pressure'
  597 = 'Delta sense' | de: 'Delta sense' | en: 'Delta sense'
  2934 = 'Delta Sense' | de: 'Delta Sense' | en: 'Delta Sense'
  461 = 'Digital'
  1557 = 'Digital Inputs' | de: 'Digital Inputs' | en: 'Digital Inputs'
  15 = 'Digital Outputs' | de: 'Digital Outputs' | en: 'Digital Outputs'
  3216 = 'display text:' | de: 'display text:' | en: 'display text:'
  3484 = 'DMC-Code:'
  548 = 'Dragon' | de: 'Dragon' | en: 'Dragon'
  3019 = 'Drehwinkel' | de: 'Drehwinkel' | en: 'Rotation angle'
  2277 = 'Drehzahl Druckpilz'
  4680 = 'Drehzahl Druckstange'
  4421 = 'Drift to initial Sense'
  6760 = 'Drive Base Position'
  169 = 'Drive Def Position'
  6603 = 'Drive Definierte Position'
  2669 = 'Drive On Pressure'
  5811 = 'Drive On Pull'
  3100 = 'Drossel' | de: 'Drossel' | en: 'Throttle'
  1539 = 'Drossel Sens Messung'
  3376 = 'Drosselwinkel' | de: 'Drosselwinkel' | en: 'Trottle angle'
  2298 = 'Drosselwinkel (Grad)' | de: 'Drosselwinkel (Grad)' | en: 'Trottle angle (Degree)'
  1404 = 'Druck' | de: 'Druck' | en: 'Pressure'
  3749 = 'Druck (PSI)' | de: 'Druck (PSI)' | en: 'Pressure (PSI)'
  4438 = 'Druckpilz'
  5892 = 'Druckstange'
  6838 = 'Druckstange Ergebnis'
  24 = 'Druckstufe (PSI/ms)' | de: 'Druckstufe (PSI/ms)' | en: 'Pressure level (PSI/ms)'
  4323 = 'Druckstück'
  528 = 'EDIT' | de: 'EDIT' | en: 'EDIT'
  667 = 'Eingabe Messprogramm'
  2331 = 'EingabeTemlegrammlänge'
  657 = 'Einheit'
  581 = 'ENABLE' | de: 'ENABLE' | en: 'ENABLE'
  1075 = 'Enable Ctrl.' | de: 'Enable Ctrl.' | en: 'Enable Ctrl.'
  216 = 'End Pressure' | de: 'End Pressure' | en: 'End Pressure'
  3120 = 'End Slope' | de: 'End Slope' | en: 'End Slope'
  706 = 'Entladen fertig' | de: 'Entladen fertig' | en: 'Entladen fertig'
  1946 = 'Error' | de: 'Error' | en: 'Error'
  1723 = 'error sum: %d' | de: 'error sum: %d' | en: 'error sum: %d'
  1256 = 'ES:' | de: 'ES:' | en: 'ES:'
  579 = 'Eventtext' | de: 'Eventtext' | en: 'Eventtext'
  342 = 'Eventtype' | de: 'Eventtype' | en: 'Eventtype'
  4374 = 'Expertmode'
  2389 = 'Expertmodus'
  3065 = 'Fahren auf Definierte Kraft'
  2520 = 'Fall 1' | de: 'Fall 1' | en: 'Fall 1'
  2479 = 'Fall 2' | de: 'Fall 2' | en: 'Fall 2'
  629 = 'Feder' | de: 'Feder' | en: 'Feder'
  1407 = 'Feeder' | de: 'Feeder' | en: 'Feeder'
  2581 = 'Fehler-Code:' | de: 'Fehler-Code:' | en: 'Error code:'
  1433 = 'Fertig zum Beladen' | de: 'Fertig zum Beladen' | en: 'Ready to load'
  840 = 'Fertig zum beladen' | de: 'Fertig zum beladen' | en: 'Ready to load'
  3850 = 'File-Path'
  196 = 'Filename'
  2245 = 'Filenamen'
  353 = 'Fox' | de: 'Fox' | en: 'Fox'
  1160 = 'Freigabe'
  838 = 'FT:' | de: 'FT:' | en: 'FT:'
  202 = 'Gain' | de: 'Gain' | en: 'Gain'
  2080 = 'Gain (PSI/ms)'
  2638 = 'Gain (PSI/ms):' | de: 'Gain (PSI/ms):' | en: 'Gain (PSI/ms):'
  1639 = 'Gain Falling 1 (PSI/ms)'
  2495 = 'Gain Falling 2 (PSI/ms)'
  5215 = 'Gain Rising (PSI/ms)'
  208 = 'Gain:' | de: 'Gain:' | en: 'Gain:'
  3301 = 'GENERAL'
  1356 = 'GET' | de: 'GET' | en: 'GET'
  1105 = 'GET INPUT REGISTER BIT' | de: 'GET INPUT REGISTER BIT' | en: 'GET INPUT REGISTER BIT'
  687 = 'GET_INPUT_REGISTER BIT' | de: 'GET_INPUT_REGISTER BIT' | en: 'GET_INPUT_REGISTER BIT'
  3276 = 'GLOBAL'
  2064 = 'GO' | de: 'GO' | en: 'GO'
  1783 = 'GRAPH' | de: 'GRAPH' | en: 'GRAPH'
  1805 = 'Graph' | de: 'Graph' | en: 'Graph'
  1418 = 'GST' | de: 'GST' | en: 'GST'
  2417 = 'Gw'
  1087 = 'HAND' | de: 'HAND' | en: 'HAND'
  1496 = 'Hauptlicht'
  2837 = 'Heat' | de: 'Heat' | en: 'Heat'
  2210 = 'HOME' | de: 'HOME' | en: 'HOME'
  1315 = 'I/Os' | de: 'I/Os' | en: 'I/Os'
  1555 = 'Increase' | de: 'Increase' | en: 'Increase'
  1549 = 'Init' | de: 'Init' | en: 'Init'
  6850 = 'INPUT MAX'
  3851 = 'INPUT MIN'
  2184 = 'IO Teil entladen' | de: 'IO Teil entladen' | en: 'Unload IO part'
  3384 = 'Ist-Geschw. (mm/s):' | de: 'Ist-Geschw. (mm/s):' | en: 'Is speed (mm/s):'
  31 = 'Ist-Position. (mm):' | de: 'Ist-Position. (mm):' | en: 'Is Position (mm):'
  5630 = 'JA'
  350 = 'JOG' | de: 'JOG' | en: 'JOG'
  846 = 'Joint Current' | de: 'Joint Current' | en: 'Joint Current'
  946 = 'Joint Mode' | de: 'Joint Mode' | en: 'Joint Mode'
  1022 = 'Joint Position' | de: 'Joint Position' | en: 'Joint Position'
  214 = 'Joint Temparatur' | de: 'Joint Temparatur' | en: 'Joint Temparatur'
  554 = 'Joint Velocitiy' | de: 'Joint Velocitiy' | en: 'Joint Velocitiy'
  543 = 'Kameraprogramm Druckpilz:'
  5774 = 'Kameraprogramm Druckstück:'
  2290 = 'KISTLER'
  872 = 'Kistler Presse'
  2961 = 'Kommando:' | de: 'Kommando:' | en: 'command:'
  1669 = 'Kontaktieren' | de: 'Kontaktieren' | en: 'contact'
  6368 = 'Kopieren'
  1354 = 'Korrekt Beladen' | de: 'Korrekt Beladen' | en: 'Correct loading'
  990 = 'Korrekt beladen' | de: 'Korrekt beladen' | en: 'Correct loading'
  163 = 'Kp: ' | de: 'Kp: ' | en: 'Kp: '
  2353 = 'Kraft'
  3173 = 'Kraft in kN:'
  998 = 'L' | de: 'L' | en: 'L'
  289 = 'Lab-Track Nb.'
  682 = 'Lab-Tracking Nb.'
  5927 = 'LabTrack Nb.'
  1107 = 'LADEN'
  6040 = 'Lampe'
  683 = 'LEC' | de: 'LEC' | en: 'LEC'
  755 = 'LED DIAG' | de: 'LED DIAG' | en: 'LED DIAG'
  411 = 'LED FAULT' | de: 'LED FAULT' | en: 'LED FAULT'
  855 = 'LED IFAULT' | de: 'LED IFAULT' | en: 'LED IFAULT'
  393 = 'LED OFAULT' | de: 'LED OFAULT' | en: 'LED OFAULT'
  845 = 'LED RUN FS' | de: 'LED RUN FS' | en: 'LED RUN FS'
  168 = 'LED RUN ST' | de: 'LED RUN ST' | en: 'LED RUN ST'
  3279 = 'Linearförderer'
  876 = 'LOAD' | de: 'LOAD' | en: 'LOAD'
  717 = 'LOAD FROM XML'
  1530 = 'Loop-Back Mode' | de: 'Loop-Back Mode' | en: 'Loop-Back Mode'
  7020 = 'Löschen'
  2596 = 'Löschen!!P5: Druckänderung in PSI'
  2074 = 'Löttemperatur:' | de: 'Löttemperatur:' | en: 'Solder temperature:'
  1207 = 'Lötzeit:' | de: 'Lötzeit:' | en: 'Solder time:'
  977 = 'm (Gain)' | de: 'm (Gain)' | en: 'm (Gain)'
  1230 = 'M380' | de: 'M380' | en: 'M380'
  605 = 'M400' | de: 'M400' | en: 'M400'
  1179 = 'M400 an Cobot 1' | de: 'M400 an Cobot 1' | en: 'M400 an Cobot 1'
  1203 = 'M400 an Cobot 2' | de: 'M400 an Cobot 2' | en: 'M400 an Cobot 2'
  186 = 'M500 an Cobot 2' | de: 'M500 an Cobot 2' | en: 'M500 an Cobot 2'
  981 = 'm=(y2-y1)/(x2-x1)' | de: 'm=(y2-y1)/(x2-x1)' | en: 'm=(y2-y1)/(x2-x1)'
  167 = 'MANUAL' | de: 'MANUAL' | en: 'MANUAL'
  4518 = 'MASCHINEN-PARAMETER'
  4836 = 'MASCHINENSPEZIFISCHE PARAMETER'
  975 = 'Max Value' | de: 'Max Value' | en: 'Max Value'
  3096 = 'Max. Current'
  2769 = 'Max. Current 1:'
  1879 = 'Max. Current 2'
  4409 = 'Max. Current 2:'
  865 = 'Max. Current in mA'
  3020 = 'Max. Current in mA:'
  2896 = 'Max. Delta to Init Sense'
  3832 = 'Max. Sense'
  1495 = 'Measure Mode' | de: 'Measure Mode' | en: 'Measure Mode'
  1479 = 'Measure Time' | de: 'Measure Time' | en: 'Measure Time'
  974 = 'Min Value' | de: 'Min Value' | en: 'Min Value'
  3171 = 'Min. Sense'
  899 = 'Mode' | de: 'Mode' | en: 'Mode'
  715 = 'Modus' | de: 'Modus' | en: 'Mode'
  610 = 'ms' | de: 'ms' | en: 'ms'
  976 = 'n (Offset)' | de: 'n (Offset)' | en: 'n (Offset)'
  982 = 'n = y1-m*x1' | de: 'n = y1-m*x1' | en: 'n = y1-m*x1'
  5506 = 'Name'
  5682 = 'Name: '
  1249 = 'NEIN'
  1718 = 'nErrCount' | de: 'nErrCount' | en: 'nErrCount'
  1707 = 'nErrId' | de: 'nErrId' | en: 'nErrId'
  527 = 'NEW' | de: 'NEW' | en: 'NEW'
  1731 = 'NIO STATION' | de: 'NIO STATION' | en: 'NIO STATION'
  4756 = 'NIO Stückzahl:'
  7555 = 'NIO Stückzahl:\t%i'
  3572 = 'NIO Stückzahl:  %i'
  315 = 'NIO Teil entladen' | de: 'NIO Teil entladen' | en: 'unload NIO part'
  5848 = 'NIO-Abwurf'
  172 = 'NO:' | de: 'NO:' | en: 'NO:'
  2977 = 'NOK' | de: 'NOK' | en: 'NOK'
  1778 = 'None' | de: 'None' | en: 'None'
  909 = 'Notaus Quittieren'
  7561 = 'num'
  842 = 'Object' | de: 'Object' | en: 'Object'
  796 = 'OFF' | de: 'OFF' | en: 'OFF'
  201 = 'Offset' | de: 'Offset' | en: 'Offset'
  207 = 'Offset:' | de: 'Offset:' | en: 'Offset:'
  532 = 'OK' | de: 'OK' | en: 'OK'
  3745 = 'OK/NOK' | de: 'OK/NOK' | en: 'OK/NOK'
  926 = 'ON' | de: 'ON' | en: 'ON'
  5008 = 'Only Cat'
  3589 = 'Only Sense'
  281 = 'OPEN' | de: 'OPEN' | en: 'OPEN'
  3678 = 'OPEN DOOR'
  1143 = 'Operator' | de: 'Operator' | en: 'Operator'
  165 = 'Out' | de: 'Out' | en: 'Out'
  5060 = 'OUTPUT MAX'
  4739 = 'OUTPUT MIN'
  993 = 'Override%' | de: 'Override%' | en: 'Override%'
  2728 = 'Overview' | de: 'Overview' | en: 'Overview'
  750 = 'P' | de: 'P' | en: 'P'
  3056 = 'P Value'
  690 = 'P1' | de: 'P1' | en: 'P1'
  5483 = 'P10: falling slope 1 max. (PSI/ms)'
  5329 = 'P10: falling slope 1 min. (PSI/ms)'
  4471 = 'P10: falling slope 1 R² min. (<1)'
  2156 = 'P10: R² Minimum (<1)'
  1309 = 'P10: Slope Fall1 Maximum'
  3123 = 'P10: Slope Fall1 Minimum'
  6037 = 'P11: falling slope 2 max. (PSI/ms)'
  421 = 'P11: falling slope 2 min. (PSI/ms)'
  5394 = 'P11: falling slope 2 R² min. (<1)'
  1170 = 'P11: R² Minimum (<1)'
  269 = 'P11: Slope Fall2 Maximum'
  1112 = 'P11: Slope Fall2 Minimum'
  3735 = 'P12: Maximaler Druckabfall in PSI'
  5342 = 'P12: Range Druck (+/- PSI)'
  1363 = 'P12: range pressure (+/- PSI)'
  2021 = 'P12: start-time check (ms)'
  294 = 'P12: Start-Zeit Kontrolle (ms)'
  2696 = 'P12: stop-time check (ms)'
  2375 = 'P12: Stop-Zeit Kontrolle (ms)'
  4607 = 'P12:max. pressuredrop (PSI)'
  1003 = 'P1: Druck Ende'
  1291 = 'P1: Druck Ende in PSI'
  2840 = 'P1: Druck Schritt'
  1876 = 'P1: Druck Schritt in PSI'
  2434 = 'P1: Druck Start'
  4514 = 'P1: Druck Start in PSI'
  5796 = 'P1: endpressure (PSI)'
  709 = 'P1: pressure-steps (PSI)'
  1663 = 'P1: startpressure (PSI)'
  447 = 'P2' | de: 'P2' | en: 'P2'
  408 = 'P2: measuretime CAT (ms)'
  1320 = 'P2: Messzeit'
  2491 = 'P2: Messzeit in ms'
  510 = 'P3' | de: 'P3' | en: 'P3'
  1269 = 'P3: Ende Messung Rising Slope'
  3917 = 'P3: Ende Messung Rising Slope in %'
  4225 = 'P3: measure end; rising slope (%)'
  2741 = 'P3: measure end; rising slope in %'
  720 = 'P4' | de: 'P4' | en: 'P4'
  996 = 'P4: measure start; rising slope (%)'
  1645 = 'P4: measure start; rising slope in %'
  2935 = 'P4: Start Messung Rising Slope in %'
  52 = 'P5' | de: 'P5' | en: 'P5'
  3441 = 'P5: Druckänderung in PSI'
  3431 = 'P5: gain (PSI/ms)'
  1979 = 'P5: rising slope deviation max. (PSI/ms)'
  5793 = 'P5: Rising Slope Deviation Max: in PSI/ms'
  5033 = 'P5: rising slope deviation min. (PSI/ms)'
  2467 = 'P5: Rising Slope Deviation Min. in PSI/ms'
  4197 = 'P5: Rising Slope Max:'
  1732 = 'P5: Rising Slope Max: in PSI/ms'
  3492 = 'P5: Rising Slope Min.'
  144 = 'P5: Rising Slope Min. in PSI/ms'
  4987 = 'P5: Rising Slope R² Min. (<1)'
  6482 = 'P5: rising slope R² Min. (<1)'
  1039 = 'P5: rising-time for const.- slope (ms)'
  3230 = 'P5: Steigungsrate in PSI/ms'
  2705 = 'P5: Zeit Steigung in ms'
  969 = 'P6' | de: 'P6' | en: 'P6'
  458 = 'P6/P7: R² Minimum (<1)'
  1851 = 'P6/P7: Slope Fall1 Maximum'
  343 = 'P6/P7: Slope Fall1 Minimum'
  2690 = 'P6: Start Falling Slope 1'
  4098 = 'P6: Start Falling Slope 1 '
  3012 = 'P6: start falling-slope 1 '
  945 = 'P7' | de: 'P7' | en: 'P7'
  3736 = 'P7: end falling-slope 1'
  4356 = 'P7: Ende Falling Slope 1'
  89 = 'P8' | de: 'P8' | en: 'P8'
  4270 = 'P8: falling slope 2 min. (PSI/ms)'
  3343 = 'P8: Start Falling Slope 2 '
  3910 = 'P9: end falling-slope 2'
  2627 = 'P9: Ende Falling Slope 2'
  928 = 'PARAMETER'
  4220 = 'Parameter'
  5646 = 'PARAMETER KOPIEREN'
  2096 = 'PARAMETER LÖSCHEN'
  1717 = 'Parameterinfo:' | de: 'Parameterinfo:' | en: 'Parameterinfo:'
  1236 = 'Parametername'
  1583 = 'Parametername:'
  6135 = 'PARAMETERSATZ LADEN'
  797 = 'Part Nb.'
  1224 = 'PB:' | de: 'PB:' | en: 'PB:'
  1480 = 'Pick and Place' | de: 'Pick and Place' | en: 'Pick and Place'
  1394 = 'Platine' | de: 'Platine' | en: 'circuit board'
  962 = 'PLC an Cobot t 1' | de: 'PLC an Cobot t 1' | en: 'PLC an Cobot t 1'
  287 = 'PLC an Cobot t 2' | de: 'PLC an Cobot t 2' | en: 'PLC an Cobot t 2'
  6164 = 'Position '
  4795 = 'Position Dreheinheit Abstützung'
  7311 = 'Position Schwe'
  1980 = 'Position Schwenkarm Druckpilz pressen'
  3601 = 'Position Schwenkarm Druckstueck pressen'
  1643 = 'Power Supply'
  882 = 'POWER SUPPLY'
  806 = 'PR' | de: 'PR' | en: 'PR'
  1162 = 'PR:' | de: 'PR:' | en: 'PR:'
  6539 = 'Pressprogamm Druckpilz:'
  2659 = 'Pressprogramm'
  6428 = 'Pressprogramm Druckstück'
  1492 = 'Pressure' | de: 'Pressure' | en: 'Pressure'
  1584 = 'PRESSURE (PSI)' | de: 'PRESSURE (PSI)' | en: 'PRESSURE (PSI)'
  3359 = 'Pressure Step' | de: 'Pressure Step' | en: 'Pressure Step'
  1065 = 'Pressure Value'
  1559 = 'Process' | de: 'Process' | en: 'Process'
  1096 = 'PRODUCT' | de: 'PRODUCT' | en: 'PRODUCT'
  3772 = 'Product' | de: 'Product' | en: 'Product'
  317 = 'Produkt' | de: 'Produkt' | en: 'Product'
  957 = 'Profinet' | de: 'Profinet' | en: 'Profinet'
  2511 = 'Projectnummer:' | de: 'Projectnummer:' | en: 'Project number:'
  849 = 'Projektnummer:' | de: 'Projektnummer:' | en: 'Project number:'
  6246 = 'Prozess'
  1889 = 'Prozess Druckpilz'
  4037 = 'Prozess Druckstange'
  3864 = 'Prozess Druckstück'
  6107 = 'PROZESS-PARAMETER'
  898 = 'PS:' | de: 'PS:' | en: 'PS:'
  1139 = 'PSI' | de: 'PSI' | en: 'PSI'
  712 = 'PW:' | de: 'PW:' | en: 'PW:'
  1399 = 'Quit' | de: 'Quit' | en: 'Quit'
  927 = 'Quit Time' | de: 'Quit Time' | en: 'Quit Time'
  82 = 'RC:' | de: 'RC:' | en: 'RC:'
  2101 = 'RcvDataHex' | de: 'RcvDataHex' | en: 'RcvDataHex'
  1497 = 'RcvDataLen' | de: 'RcvDataLen' | en: 'RcvDataLen'
  2648 = 'RcvDataStr' | de: 'RcvDataStr' | en: 'RcvDataStr'
  628 = 'RD:' | de: 'RD:' | en: 'RD:'
  1823 = 'READ' | de: 'READ' | en: 'READ'
  520 = 'read_output_boolean_register(address)' | de: 'read_output_boolean_register(address)' | en: 'read_output_boolean_register(address)'
  3937 = 'Referenzfahrt'
  90 = 'Referezanfahren'
  1099 = 'REGISTER' | de: 'REGISTER' | en: 'REGISTER'
  228 = 'Regler' | de: 'Regler' | en: 'Rulings'
  2804 = 'Relativ' | de: 'Relativ' | en: 'Relativ'
  4041 = 'REMOTE AKTIV'
  1777 = 'Repeat counter sens-testing'
  575 = 'Repeat counter sensing'
  6055 = 'repeat-counter sens-testing'
  622 = 'RES:' | de: 'RES:' | en: 'RES:'
  4984 = 'Reserve'
  1561 = 'Reset' | de: 'Reset' | en: 'Reset'
  678 = 'RESET' | de: 'RESET' | en: 'RESET'
  480 = 'Reset Counters' | de: 'Reset Counters' | en: 'Reset Counters'
  7531 = 'Reset NIO Stückzahl'
  212 = 'RESTORE' | de: 'RESTORE' | en: 'RESTORE'
  247 = 'RESULT' | de: 'RESULT' | en: 'RESULT'
  3657 = 'Result' | de: 'Result' | en: 'Result'
  3249 = 'RESULT TABLE'
  3207 = 'Result Table'
  2800 = 'Retest'
  2582 = 'rise time:'
  761 = 'Robot' | de: 'Robot' | en: 'Robot'
  891 = 'Robot current:' | de: 'Robot current:' | en: 'Robot current:'
  1210 = 'Robot mode:' | de: 'Robot mode:' | en: 'Robot mode:'
  1094 = 'Robot/Safety' | de: 'Robot/Safety' | en: 'Robot/Safety'
  5663 = 'rpm'
  3789 = 'RQ' | de: 'RQ' | en: 'RQ'
  5373 = 'RQ-Nb.'
  2785 = 'RQ-Nr.' | de: 'RQ-Nr.' | en: 'RQ-Nr.'
  2577 = 'RQ-Number' | de: 'RQ-Number' | en: 'RQ-Number'
  822 = 'RQ-NUMBER' | de: 'RQ-NUMBER' | en: 'RQ-NUMBER'
  2313 = 'RQ-Nummer' | de: 'RQ-Nummer' | en: 'RQ-Nummer'
  288 = 'R²' | de: 'R²' | en: 'R²'
  2327 = 'R² (Falling 1):'
  3658 = 'R² (Falling 2):'
  1021 = 'R² (Risin):'
  2539 = 'R² (Rising):'
  5704 = 'R² Slope Fall 1'
  2363 = 'R² Slope Fall 2'
  4675 = 'R² Slope Rise'
  2046 = 'R²:' | de: 'R²:' | en: 'R²:'
  1023 = 'Rückgabe:' | de: 'Rückgabe:' | en: 'Return:'
  847 = 'Safety Mode:' | de: 'Safety Mode:' | en: 'Safety Mode:'
  211 = 'SAVE' | de: 'SAVE' | en: 'SAVE'
  116 = 'SAVE NEW'
  2222 = 'SAVE TO XML'
  526 = 'SCALED' | de: 'SCALED' | en: 'SCALED'
  531 = 'SCALED:' | de: 'SCALED:' | en: 'SCALED:'
  3727 = 'Scannen'
  6736 = 'Scanner aktivieren'
  5592 = 'SCHLIESSEN'
  2496 = 'Schließen'
  2462 = 'Schott'
  2752 = 'Schrittmotor Druckpilz'
  1746 = 'Schrittmotor Druckstange'
  5142 = 'Schrittmotor Schwenkarm'
  4866 = 'Schutztür verriegeln'
  3872 = 'Schwenk-\nantrieb'
  2802 = 'Schwenkantrieb'
  2455 = 'Schwenklippe'
  8007 = 'Schwingförderer'
  3268 = 'SEARCH RQ AND LOAD PARAMETER'
  1482 = 'SELECT ALL' | de: 'SELECT ALL' | en: 'SELECT ALL'
  2155 = 'SELECT NONE' | de: 'SELECT NONE' | en: 'SELECT NONE'
  708 = 'Select Parameter'
  1586 = 'Send' | de: 'Send' | en: 'Send'
  1537 = 'Sense' | de: 'Sense' | en: 'Sense'
  1756 = 'Sense After' | de: 'Sense After' | en: 'Sense After'
  3172 = 'Sense initial'
  2201 = 'Sense Measure' | de: 'Sense Measure' | en: 'Sense Measure'
  1815 = 'Sense-Test'
  4280 = 'Sensor 1'
  5170 = 'Sensor 2'
  1355 = 'SEPERATOR' | de: 'SEPERATOR' | en: 'SEPERATOR'
  989 = 'Seperator' | de: 'Seperator' | en: 'Seperator'
  1000 = 'SERIAL' | de: 'SERIAL' | en: 'SERIAL'
  2114 = 'Serial' | de: 'Serial' | en: 'Serial'
  1698 = 'Serial COM' | de: 'Serial COM' | en: 'Serial COM'
  148 = 'SerialCom.aRcvDataHex[INDEX]' | de: 'SerialCom.aRcvDataHex[INDEX]' | en: 'SerialCom.aRcvDataHex[INDEX]'
  1518 = 'SerialCom.aRcvDataLen[INDEX]' | de: 'SerialCom.aRcvDataLen[INDEX]' | en: 'SerialCom.aRcvDataLen[INDEX]'
  630 = 'SerialCom.aRcvDataStr[INDEX]' | de: 'SerialCom.aRcvDataStr[INDEX]' | en: 'SerialCom.aRcvDataStr[INDEX]'
  1712 = 'sErrSource' | de: 'sErrSource' | en: 'sErrSource'
  2078 = 'Service' | de: 'Service' | en: 'Service'
  215 = 'SES:' | de: 'SES:' | en: 'SES:'
  1437 = 'SET' | de: 'SET' | en: 'SET'
  2364 = 'Set' | de: 'Set' | en: 'Set'
  2610 = 'Set Position' | de: 'Set Position' | en: 'Set Position'
  3311 = 'Set Slope' | de: 'Set Slope' | en: 'Set Slope'
  164 = 'Setpoint' | de: 'Setpoint' | en: 'Setpoint'
  5233 = 'Setpoint P'
  1282 = 'Setpoint Pressure'
  2257 = 'Setpoint Pressure (PSI):'
  405 = 'setpoint pressure:' | de: 'setpoint pressure:' | en: 'setpoint pressure:'
  2989 = 'Setpoint PSI'
  3033 = 'Setpoint Slope' | de: 'Setpoint Slope' | en: 'Setpoint Slope'
  2791 = 'Setpoint:' | de: 'Setpoint:' | en: 'Setpoint:'
  320 = 'Shuttle' | de: 'Shuttle' | en: 'Shuttle'
  1313 = 'Slope' | de: 'Slope' | en: 'Slope'
  1995 = 'SLOPE' | de: 'SLOPE' | en: 'SLOPE'
  463 = 'Slope (PSI/ms)' | de: 'Slope (PSI/ms)' | en: 'Slope (PSI/ms)'
  2551 = 'SLOPE (PSI/ms)' | de: 'SLOPE (PSI/ms)' | en: 'SLOPE (PSI/ms)'
  44 = 'Slope calibrate range max:'
  1656 = 'Slope calibrate range mIN:'
  2086 = 'Slope calibrate range min:'
  1683 = 'Slope Fall' | de: 'Slope Fall' | en: 'Slope Fall'
  3017 = 'Slope Fall 1'
  4703 = 'Slope Fall 1 R²'
  4609 = 'Slope Fall 1 Value'
  2976 = 'Slope Fall 2' | de: 'Slope Fall 2' | en: 'Slope Fall 2'
  5956 = 'Slope Fall 2 R²'
  3787 = 'Slope Fall 2 Value'
  1335 = 'Slope Rise'
  2706 = 'Slope Rise R²'
  1222 = 'Slope Rise Set'
  1861 = 'Slope Rise Setpoint'
  2621 = 'Slope Rise Value'
  2818 = 'Slope Settings'
  1603 = 'Slope Step' | de: 'Slope Step' | en: 'Slope Step'
  3776 = 'Slope-Test'
  2185 = 'Slope:'
  4229 = 'SLOPE: ' | de: 'SLOPE: ' | en: 'SLOPE: '
  1307 = 'SMC' | de: 'SMC' | en: 'SMC'
  1900 = 'Soll der ausgewählte Parametersatz gelöscht werden?'
  2400 = 'SORTIEREN' | de: 'SORTIEREN' | en: 'SORT'
  385 = 'SS:' | de: 'SS:' | en: 'SS:'
  244 = 'ST:' | de: 'ST:' | en: 'ST:'
  351 = 'START' | de: 'START' | en: 'START'
  222 = 'Start Before' | de: 'Start Before' | en: 'Start Before'
  677 = 'Start Pressure' | de: 'Start Pressure' | en: 'Start Pressure'
  3254 = 'Start Slope' | de: 'Start Slope' | en: 'Start Slope'
  897 = 'Start Time' | de: 'Start Time' | en: 'Start Time'
  2381 = 'StartSlope' | de: 'StartSlope' | en: 'StartSlope'
  1665 = 'Startwert Auswertung Druckpilz'
  1090 = 'Startwert Auswertung Druckstange'
  4012 = 'Static Throttle Angle'
  1543 = 'Status' | de: 'Status' | en: 'Status'
  6757 = 'Status fügen'
  791 = 'Steilförderer'
  5200 = 'Stop'
  1833 = 'Strat Time'
  25 = 'Taktzeit' | de: 'Taktzeit' | en: 'Cycle time'
  2172 = 'TANK' | de: 'TANK' | en: 'TANK'
  124 = 'TB:' | de: 'TB:' | en: 'TB:'
  230 = 'TCP Force' | de: 'TCP Force' | en: 'TCP Force'
  1131 = 'TCP Position' | de: 'TCP Position' | en: 'TCP Position'
  988 = 'TCP Torque' | de: 'TCP Torque' | en: 'TCP Torque'
  614 = 'TCP Velocitiy' | de: 'TCP Velocitiy' | en: 'TCP Velocitiy'
  160 = 'Td: ' | de: 'Td: ' | en: 'Td: '
  290 = 'Telegrammlänge Presse'
  1516 = 'Teller' | de: 'Teller' | en: 'Plate'
  1247 = 'Temp Value'
  3655 = 'Temp.' | de: 'Temp.' | en: 'Temp.'
  6088 = 'Temp. Value'
  2062 = 'Temperartur' | de: 'Temperartur' | en: 'Temperature'
  3628 = 'Temperatur' | de: 'Temperatur' | en: 'Temperature'
  5165 = 'Temperature Maximum'
  1244 = 'temperature maximum'
  3942 = 'Temperature Minimum'
  3698 = 'temperature minimum'
  3423 = 'Test Mode' | de: 'Test Mode' | en: 'Test Mode'
  4770 = 'Testpressure'
  45 = 'Text' | de: 'Text' | en: 'Text'
  2421 = 'Text:' | de: 'Text:' | en: 'Text:'
  452 = 'Throttle' | de: 'Throttle' | en: 'Throttle'
  1971 = 'Throttle Angle Table'
  4580 = 'Throttle angle:'
  3392 = 'throttle degree for sensing: '
  735 = 'Throttle Setpoint' | de: 'Throttle Setpoint' | en: 'Throttle Setpoint'
  229 = 'Throttle Value' | de: 'Throttle Value' | en: 'Throttle Value'
  1301 = 'Time' | de: 'Time' | en: 'Time'
  1836 = 'TIPP' | de: 'TIPP' | en: 'TIPP'
  1964 = 'TIPPEN' | de: 'TIPPEN' | en: 'TIPPEN'
  801 = 'Tn: ' | de: 'Tn: ' | en: 'Tn: '
  1485 = 'Tool analog out' | de: 'Tool analog out' | en: 'Tool analog out'
  318 = 'Tool Current' | de: 'Tool Current' | en: 'Tool Current'
  585 = 'Tool Current [mA]' | de: 'Tool Current [mA]' | en: 'Tool Current [mA]'
  55 = 'Tool Inputs' | de: 'Tool Inputs' | en: 'Tool Inputs'
  6170 = 'Tool Kamera Bohrung Anwesenheit'
  5319 = 'Tool Kamera Bohrung Druckpilz'
  6251 = 'Tool Kamera Bohrung Druckstange'
  4273 = 'Tool Kamera Druckstange anwesenheit'
  3222 = 'Tool Kamera Druckstange Anwesenheit'
  195 = 'Tool Outputs' | de: 'Tool Outputs' | en: 'Tool Outputs'
  1250 = 'Tool Voltage' | de: 'Tool Voltage' | en: 'Tool Voltage'
  1607 = 'Tool Voltage [V]' | de: 'Tool Voltage [V]' | en: 'Tool Voltage [V]'
  226 = 'Tray' | de: 'Tray' | en: 'Tray'
  5788 = 'Trigger'
  802 = 'Tv: ' | de: 'Tv: ' | en: 'Tv: '
  1027 = 'TXT'
  1358 = 'Typ Daimler' | de: 'Typ Daimler' | en: 'Typ Daimler'
  225 = 'Typ Dragon' | de: 'Typ Dragon' | en: 'Typ Dragon'
  719 = 'Typ Fox' | de: 'Typ Fox' | en: 'Typ Fox'
  5697 = 'TYP-SPEZIFISCHE PARAMETER'
  2497 = 'TYPSPEZIFISCHE PARAMETER'
  525 = 'UNSCALED' | de: 'UNSCALED' | en: 'UNSCALED'
  6412 = 'UNSCALED OUTPUT'
  530 = 'UNSCALED:' | de: 'UNSCALED:' | en: 'UNSCALED:'
  3440 = 'UPV'
  1965 = 'UPV Channel'
  4757 = 'UPV Clock Freqence'
  4428 = 'UPV Clock Freqence inHz'
  4804 = 'UPV Fequence'
  913 = 'UPV Impendance'
  2742 = 'UPV Logic Voltage'
  1353 = 'UPV Logic Voltage in ??'
  3306 = 'UPV Logic Voltage in mV'
  5839 = 'UPV Logic Voltage in V'
  2127 = 'UPV Voltage'
  4190 = 'UPV Voltage in mV:'
  566 = 'Vac' | de: 'Vac' | en: 'Vac'
  947 = 'VAC' | de: 'VAC' | en: 'VAC'
  5537 = 'Vakuum-Pumpe'
  1193 = 'VALUE' | de: 'VALUE' | en: 'VALUE'
  1864 = 'Value' | de: 'Value' | en: 'Value'
  204 = 'Value Max' | de: 'Value Max' | en: 'Value Max'
  210 = 'Value Max:' | de: 'Value Max:' | en: 'Value Max:'
  203 = 'Value Min' | de: 'Value Min' | en: 'Value Min'
  209 = 'Value Min:' | de: 'Value Min:' | en: 'Value Min:'
  206 = 'Value Scale' | de: 'Value Scale' | en: 'Value Scale'
  205 = 'Value Unscale' | de: 'Value Unscale' | en: 'Value Unscale'
  534 = 'Value:' | de: 'Value:' | en: 'Value:'
  3888 = 'VDD 1'
  5573 = 'VDD 2'
  4989 = 'VDD1'
  3962 = 'VDD2'
  84 = 'Vereinzeler' | de: 'Vereinzeler' | en: 'Seperator'
  1538 = 'Vereinzelung' | de: 'Vereinzelung' | en: 'Isolation'
  110 = 'Vereinzelung/Roboter' | de: 'Vereinzelung/Roboter' | en: 'Isolation/Robot'
  3200 = 'Versatzwinkel Druckpilz'
  900 = 'Versatzwinkel Druckstange'
  3329 = 'Vibrationsbunker'
  824 = 'VIRTU' | de: 'VIRTU' | en: 'VIRTU'
  197 = 'virtual input' | de: 'virtual input' | en: 'virtual input'
  662 = 'VIRTUAL INPUT 0-31' | de: 'VIRTUAL INPUT 0-31' | en: 'VIRTUAL INPUT 0-31'
  782 = 'VIRTUAL INPUT 0-31:  ' | de: 'VIRTUAL INPUT 0-31:  ' | en: 'VIRTUAL INPUT 0-31:  '
  601 = 'VIRTUAL INPUT 32-63:  ' | de: 'VIRTUAL INPUT 32-63:  ' | en: 'VIRTUAL INPUT 32-63:  '
  423 = 'VIRTUAL INPUT 64-95:  ' | de: 'VIRTUAL INPUT 64-95:  ' | en: 'VIRTUAL INPUT 64-95:  '
  17 = 'VIRTUAL INPUT 96-127:  ' | de: 'VIRTUAL INPUT 96-127:  ' | en: 'VIRTUAL INPUT 96-127:  '
  29 = 'VIRTUAL OUTPUT 0-31:  ' | de: 'VIRTUAL OUTPUT 0-31:  ' | en: 'VIRTUAL OUTPUT 0-31:  '
  325 = 'VIRTUAL OUTPUT 32-63:  ' | de: 'VIRTUAL OUTPUT 32-63:  ' | en: 'VIRTUAL OUTPUT 32-63:  '
  887 = 'VIRTUAL OUTPUT 64-95:  ' | de: 'VIRTUAL OUTPUT 64-95:  ' | en: 'VIRTUAL OUTPUT 64-95:  '
  825 = 'VIRTUAL OUTPUT 96-127:  ' | de: 'VIRTUAL OUTPUT 96-127:  ' | en: 'VIRTUAL OUTPUT 96-127:  '
  264 = 'VL:' | de: 'VL:' | en: 'VL:'
  4271 = 'Voltage'
  2134 = 'Voltage 1'
  2052 = 'Voltage 1:'
  2926 = 'Voltage 2'
  2798 = 'Voltage in V:'
  131 = 'VON: '
  673 = 'Vorheizzeit:' | de: 'Vorheizzeit:' | en: 'Preheat time:'
  3137 = 'Vorschub +' | de: 'Vorschub +' | en: 'Feed +'
  2312 = 'Vorschub -' | de: 'Vorschub -' | en: 'Feed -'
  337 = 'Vorschubgeschw.:' | de: 'Vorschubgeschw.:' | en: 'Feed rate.:'
  4091 = 'Votage 2:'
  5938 = 'Weg in mm:'
  3253 = 'Wert'
  1038 = 'Winkel Drossel in °:' | de: 'Winkel Drossel in °:' | en: 'Angle throttle in °:'
  1041 = 'Winkel Drossel:' | de: 'Winkel Drossel:' | en: 'Angle throttle:'
  1595 = 'Winkelversatz Druckpilz:'
  3452 = 'Winkelversatz Druckstange:'
  795 = 'WORK' | de: 'WORK' | en: 'WORK'
  1550 = 'WRITE' | de: 'WRITE' | en: 'WRITE'
  800 = 'write_input_boolean_register(address, value)' | de: 'write_input_boolean_register(address, value)' | en: 'write_input_boolean_register(address, value)'
  484 = 'write_input_float_register(address, value)' | de: 'write_input_float_register(address, value)' | en: 'write_input_float_register(address, value)'
  1749 = 'write_input_integer_register(address, value)  ' | de: 'write_input_integer_register(address, value)  ' | en: 'write_input_integer_register(address, value)  '
  818 = 'write_output_boolean_register(address, value)' | de: 'write_output_boolean_register(address, value)' | en: 'write_output_boolean_register(address, value)'
  561 = 'write_output_float_register(address, value)' | de: 'write_output_float_register(address, value)' | en: 'write_output_float_register(address, value)'
  1359 = 'write_output_integer_register(address, value)  ' | de: 'write_output_integer_register(address, value)  ' | en: 'write_output_integer_register(address, value)  '
  983 = 'X' | de: 'X' | en: 'X'
  979 = 'x (Unscaled)' | de: 'x (Unscaled)' | en: 'x (Unscaled)'
  567 = 'XX' | de: 'XX' | en: 'XX'
  978 = 'y (Scaled)' | de: 'y (Scaled)' | en: 'y (Scaled)'
  980 = 'y=m*x+n' | de: 'y=m*x+n' | en: 'y=m*x+n'
  1141 = 'Zeit Nachtemperieren:' | de: 'Zeit Nachtemperieren:' | en: 'Zeit Nachtemperieren:'
  635 = 'Zusatzinfo' | de: 'Zusatzinfo' | en: 'Zusatzinfo'
  6903 = '°'
  5487 = '° (Grad)'
  3912 = 'Übernehmen'
END_TEXTLIST

// ---- MODULE/ACTOR_VALVE/PNEUMATIC_ACTOR/TXTLIST/TXT_LIST_PNEMATIC_ACTOR.TcTLO
TEXTLIST TXT_LIST_PNEMATIC_ACTOR
  1 = 'Timeout: Bewegung nach Arbeitsstellung' | de: 'Timeout: Bewegung nach Arbeitsstellung' | en: 'Timeout: Move to Workposition'
  2 = 'Timeout: Bewegung nach Grundstellung' | de: 'Timeout: Bewegung nach Grundstellung' | en: 'Timeout: Move to Basepostion'
  3 = 'fährt in Grundposition' | de: 'fährt in Grundposition' | en: 'moves to Baseposition'
  4 = 'ist in Grundposition' | de: 'ist in Grundposition' | en: 'in Baseposition'
  5 = 'fährt in Arbeitsposition' | de: 'fährt in Arbeitsposition' | en: 'moves to Workposition'
  6 = 'ist in Arbeitsposition' | de: 'ist in Arbeitsposition' | en: 'in Workposition'
  7 = 'in undefinierter Position' | de: 'in undefinierter Position' | en: 'in undefined postion'
  8 = 'Timeout bei Fahrt nach Grundstellung' | de: 'Timeout bei Fahrt nach Grundstellung' | en: 'Timeout: Move to Basepos.'
  9 = 'Timeout bei Fahrt nach Arbeitsstellung' | de: 'Timeout bei Fahrt nach Arbeitsstellung' | en: 'Timeout: Move to Workpos.'
  11 = 'Vakuum ein / Druck nicht erreicht' | de: 'Vakuum ein / Druck nicht erreicht' | en: 'vaccum on / pressure NOK'
  12 = 'Vakuum ein / Druck OK' | de: 'Vakuum ein / Druck OK' | en: 'vaccum on / pressure OK'
  13 = 'Abblasen ein' | de: 'Abblasen ein' | en: 'blow out'
  14 = 'nicht aktiv' | de: 'nicht aktiv' | en: 'not active'
  15 = 'ist in Mittelstellung' | de: 'ist in Mittelstellung' | en: 'in mid position'
  16 = 'blockiert durch' | de: 'blockiert durch' | en: 'locked by'
   = ''
END_TEXTLIST

// ---- MODULE/ACTOR_VALVE/PNEUMATIC_ACTOR/VISU/VisuCylinderGripperDown.TcVIS
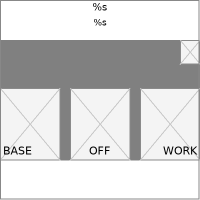
VISUALIZATION VisuCylinderGripperDown  // 200x200
VAR_IN_OUT
	fbVisuCylinder: FB_VISU_CYLINDER;
END_VAR
    Textfield (0,15 200x15), "%s", text variable: fbVisuCylinder.strInfo, colour toggle: fbVisuCylinder.stEvent.bEventActive
    Textfield (0,0 200x14), "%s", text variable: fbVisuCylinder.strFullObjName
    Group (40,40 120x80)
        OnMouseClick: execute { fbVisuCylinder.bFrameInvisible:=false; }
        RoundedRectangle (85,30 20x50)
            p3560616238: fbVisuCylinder.iMoveSmall
        RoundedRectangle (5,30 20x50)
            p3560616238: fbVisuCylinder.iNegMoveSmall
        RoundedRectangle (0,20 110x20)
        Rectangle (0,0 110x45)
    Group (70,125 60x30)
        Image (0,0 30x30), invisible if: fbVisuCylinder.bWorkArrowInvisible, image: VisuSymbols.Symbols.ArrowBoldRight
            p2175578022: fbVisuCylinder.dwFrameColorWork
        Image (30,0 30x30), invisible if: fbVisuCylinder.bWorkArrowInvisible, image: VisuSymbols.Symbols.ArrowBoldLeft
            p2175578022: fbVisuCylinder.dwFrameColorWork
    Group (70,125 60x30)
        Image (0,0 30x30), invisible if: fbVisuCylinder.bBaseArrowInvisible, image: VisuSymbols.Symbols.ArrowBoldLeft
            p2175578022: fbVisuCylinder.dwFrameColorBase
        Image (30,0 30x30), invisible if: fbVisuCylinder.bBaseArrowInvisible, image: VisuSymbols.Symbols.ArrowBoldRight
            p2175578022: fbVisuCylinder.dwFrameColorBase
    Frame (0,40 200x120), invisible if: fbVisuCylinder.bFrameInvisible, frame switch variable: fbVisuCylinder.iFrame
        shows VisuCylinderHorRightCtrl(fbVisuCylinder := fbVisuCylinder)
END_VISUALIZATION

